LIN {X 0.253,Y -606.184,Z 1339.063,A 0.000,B 0.000,C 90.000,E1 47.391} C_DIS
LIN {X 0.399,Y -606.408,Z 1339.055,A 0.000,B 0.000,C 90.000,E1 45.810} C_DIS
LIN {X 0.066,Y -606.395,Z 1339.049,A 0.000,B 0.000,C 90.000,E1 44.798} C_DIS
LIN {X -0.075,Y -606.253,Z 1339.045,A 0.000,B 0.000,C 90.000,E1 44.028} C_DIS
LIN {X 0.206,Y -605.996,Z 1339.040,A 0.000,B 0.000,C 90.000,E1 43.218} C_DIS
LIN {X -0.072,Y -605.394,Z 1339.031,A 0.000,B 0.000,C 90.000,E1 41.676} C_DIS
LIN {X -0.161,Y -604.795,Z 1339.024,A 0.000,B 0.000,C 90.000,E1 40.378} C_DIS
LIN {X 0.075,Y -603.985,Z 1339.016,A 0.000,B 0.000,C 90.000,E1 38.785} C_DIS
LIN {X 0.122,Y -603.759,Z 1339.013,A 0.000,B 0.000,C 90.000,E1 38.257} C_DIS
LIN {X 0.089,Y -602.680,Z 1339.005,A 0.000,B 0.000,C 90.000,E1 36.950} C_DIS
LIN {X -0.224,Y -601.348,Z 1339.000,A 0.000,B 0.000,C 90.000,E1 35.931} C_DIS
LIN {X -0.077,Y -599.648,Z 1338.994,A 0.000,B 0.000,C 90.000,E1 34.865} C_DIS
LIN {X -0.395,Y -597.109,Z 1338.986,A 0.000,B 0.000,C 90.000,E1 33.579} C_DIS
LIN {X -0.042,Y -595.373,Z 1338.982,A 0.000,B 0.000,C 90.000,E1 32.752} C_DIS
LIN {X -0.025,Y -593.352,Z 1338.978,A 0.000,B 0.000,C 90.000,E1 31.957} C_DIS
LIN {X 0.082,Y -591.844,Z 1338.975,A 0.000,B 0.000,C 90.000,E1 31.416} C_DIS
LIN {X 0.258,Y -588.410,Z 1338.969,A 0.000,B 0.000,C 90.000,E1 30.335} C_DIS
LIN {X 0.204,Y -585.387,Z 1338.964,A 0.000,B 0.000,C 90.000,E1 29.539} C_DIS
LIN {X -0.037,Y -583.137,Z 1338.961,A 0.000,B 0.000,C 90.000,E1 29.027} C_DIS
LIN {X -0.212,Y -578.917,Z 1338.956,A 0.000,B 0.000,C 90.000,E1 28.103} C_DIS
LIN {X 0.212,Y -575.437,Z 1338.952,A 0.000,B 0.000,C 90.000,E1 27.385} C_DIS
LIN {X -0.253,Y -570.967,Z 1338.948,A 0.000,B 0.000,C 90.000,E1 26.616} C_DIS
LIN {X -0.161,Y -566.910,Z 1338.944,A 0.000,B 0.000,C 90.000,E1 25.924} C_DIS
LIN {X 0.139,Y -562.460,Z 1338.940,A 0.000,B 0.000,C 90.000,E1 25.207} C_DIS
LIN {X -0.057,Y -555.714,Z 1338.935,A 0.000,B 0.000,C 90.000,E1 24.259} C_DIS
LIN {X -0.045,Y -547.161,Z 1338.929,A 0.000,B 0.000,C 90.000,E1 23.153} C_DIS
LIN {X -0.036,Y -542.466,Z 1338.926,A 0.000,B 0.000,C 90.000,E1 22.589} C_DIS
LIN {X 0.115,Y -532.861,Z 1338.919,A 0.000,B 0.000,C 90.000,E1 21.482} C_DIS
LIN {X 0.055,Y -525.225,Z 1338.915,A 0.000,B 0.000,C 90.000,E1 20.663} C_DIS
LIN {X -0.228,Y -513.411,Z 1338.908,A 0.000,B 0.000,C 90.000,E1 19.450} C_DIS
LIN {X -0.010,Y -502.802,Z 1338.902,A 0.000,B 0.000,C 90.000,E1 18.308} C_DIS
LIN {X -0.186,Y -495.880,Z 1338.898,A 0.000,B 0.000,C 90.000,E1 17.638} C_DIS
LIN {X 0.077,Y -491.962,Z 1338.896,A 0.000,B 0.000,C 90.000,E1 17.221} C_DIS
LIN {X 0.076,Y -479.200,Z 1338.889,A 0.000,B 0.000,C 90.000,E1 16.024} C_DIS
LIN {X 0.163,Y -470.528,Z 1338.885,A 0.000,B 0.000,C 90.000,E1 15.190} C_DIS
LIN {X -0.090,Y -457.861,Z 1338.878,A 0.000,B 0.000,C 90.000,E1 14.008} C_DIS
LIN {X -0.116,Y -440.530,Z 1338.868,A 0.000,B 0.000,C 90.000,E1 12.299} C_DIS
LIN {X -0.086,Y -423.447,Z 1338.858,A 0.000,B 0.000,C 90.000,E1 10.489} C_DIS
LIN {X 0.042,Y -408.056,Z 1338.849,A 0.000,B 0.000,C 90.000,E1 8.746} C_DIS
LIN {X 0.112,Y -399.560,Z 1338.843,A 0.000,B 0.000,C 90.000,E1 7.757} C_DIS
LIN {X -0.011,Y -396.193,Z 1338.841,A 0.000,B 0.000,C 90.000,E1 7.352} C_DIS
LIN {X -0.095,Y -395.192,Z 1338.840,A 0.000,B 0.000,C 90.000,E1 7.182} C_DIS
LIN {X -0.159,Y -394.889,Z 1338.839,A 0.000,B 0.000,C 90.000,E1 7.125} C_DIS
LIN {X -0.197,Y -394.881,Z 1338.839,A 0.000,B 0.000,C 90.000,E1 7.125} C_DIS
LIN {X 0.156,Y -394.888,Z 1338.839,A 0.000,B 0.000,C 90.000,E1 7.068} C_DIS
LIN {X 0.119,Y -394.922,Z 1338.839,A 0.000,B 0.000,C 90.000,E1 7.068} C_DIS
LIN {X -0.088,Y -395.768,Z 1338.839,A 0.000,B 0.000,C 90.000,E1 7.004} C_DIS
LIN {X 0.079,Y -399.281,Z 1338.837,A 0.000,B 0.000,C 90.000,E1 6.663} C_DIS
LIN {X -0.111,Y -407.017,Z 1338.834,A 0.000,B 0.000,C 90.000,E1 6.144} C_DIS
LIN {X 0.037,Y -415.213,Z 1338.831,A 0.000,B 0.000,C 90.000,E1 5.568} C_DIS
LIN {X 0.038,Y -416.883,Z 1338.830,A 0.000,B 0.000,C 90.000,E1 5.454} C_DIS
LIN {X -0.059,Y -423.003,Z 1338.828,A 0.000,B 0.000,C 90.000,E1 4.992} C_DIS
LIN {X -0.215,Y -430.404,Z 1338.824,A 0.000,B 0.000,C 90.000,E1 4.359} C_DIS
LIN {X 0.191,Y -439.080,Z 1338.819,A 0.000,B 0.000,C 90.000,E1 3.440} C_DIS
LIN {X -0.097,Y -443.387,Z 1338.817,A 0.000,B 0.000,C 90.000,E1 3.037} C_DIS
LIN {X 0.196,Y -450.196,Z 1338.813,A 0.000,B 0.000,C 90.000,E1 2.236} C_DIS
LIN {X -0.176,Y -455.607,Z 1338.809,A 0.000,B 0.000,C 90.000,E1 1.661} C_DIS
LIN {X 0.189,Y -461.755,Z 1338.805,A 0.000,B 0.000,C 90.000,E1 0.859} C_DIS
LIN {X 0.147,Y -466.546,Z 1338.801,A 0.000,B 0.000,C 90.000,E1 0.229} C_DIS
LIN {X 0.070,Y -473.059,Z 1338.796,A 0.000,B 0.000,C 90.000,E1 359.312} C_DIS
LIN {X -0.233,Y -478.042,Z 1338.792,A 0.000,B 0.000,C 90.000,E1 358.568} C_DIS
LIN {X 0.005,Y -482.684,Z 1338.788,A 0.000,B 0.000,C 90.000,E1 357.764} C_DIS
LIN {X -0.217,Y -486.975,Z 1338.783,A 0.000,B 0.000,C 90.000,E1 357.020} C_DIS
LIN {X -0.048,Y -490.251,Z 1338.780,A 0.000,B 0.000,C 90.000,E1 356.388} C_DIS
LIN {X -0.173,Y -493.903,Z 1338.776,A 0.000,B 0.000,C 90.000,E1 355.641} C_DIS
LIN {X -0.093,Y -497.944,Z 1338.771,A 0.000,B 0.000,C 90.000,E1 354.723} C_DIS
LIN {X -0.099,Y -501.093,Z 1338.766,A 0.000,B 0.000,C 90.000,E1 353.970} C_DIS
LIN {X 0.187,Y -503.472,Z 1338.763,A 0.000,B 0.000,C 90.000,E1 353.337} C_DIS
LIN {X -0.014,Y -505.647,Z 1338.760,A 0.000,B 0.000,C 90.000,E1 352.761} C_DIS
LIN {X 0.195,Y -509.626,Z 1338.753,A 0.000,B 0.000,C 90.000,E1 351.546} C_DIS
LIN {X -0.008,Y -512.111,Z 1338.748,A 0.000,B 0.000,C 90.000,E1 350.679} C_DIS
LIN {X -0.125,Y -515.124,Z 1338.742,A 0.000,B 0.000,C 90.000,E1 349.511} C_DIS
LIN {X -0.180,Y -517.123,Z 1338.737,A 0.000,B 0.000,C 90.000,E1 348.634} C_DIS
LIN {X -0.221,Y -519.485,Z 1338.730,A 0.000,B 0.000,C 90.000,E1 347.465} C_DIS
LIN {X -0.114,Y -521.403,Z 1338.724,A 0.000,B 0.000,C 90.000,E1 346.284} C_DIS
LIN {X -0.110,Y -522.626,Z 1338.719,A 0.000,B 0.000,C 90.000,E1 345.408} C_DIS
LIN {X 0.031,Y -523.577,Z 1338.714,A 0.000,B 0.000,C 90.000,E1 344.519} C_DIS
LIN {X 0.181,Y -524.262,Z 1338.709,A 0.000,B 0.000,C 90.000,E1 343.630} C_DIS
LIN {X -0.012,Y -524.796,Z 1338.704,A 0.000,B 0.000,C 90.000,E1 342.779} C_DIS
LIN {X 0.146,Y -524.986,Z 1338.700,A 0.000,B 0.000,C 90.000,E1 341.891} C_DIS
LIN {X 0.131,Y -524.847,Z 1338.693,A 0.000,B 0.000,C 90.000,E1 340.732} C_DIS
LIN {X 0.119,Y -524.172,Z 1338.687,A 0.000,B 0.000,C 90.000,E1 339.571} C_DIS
LIN {X -0.067,Y -523.171,Z 1338.682,A 0.000,B 0.000,C 90.000,E1 338.720} C_DIS
LIN {X -0.231,Y -522.344,Z 1338.679,A 0.000,B 0.000,C 90.000,E1 338.156} C_DIS
LIN {X 0.086,Y -521.302,Z 1338.675,A 0.000,B 0.000,C 90.000,E1 337.539} C_DIS
LIN {X 0.240,Y -520.884,Z 1338.674,A 0.000,B 0.000,C 90.000,E1 337.230} C_DIS
LIN {X 0.211,Y -519.215,Z 1338.669,A 0.000,B 0.000,C 90.000,E1 336.357} C_DIS
LIN {X 0.164,Y -517.178,Z 1338.664,A 0.000,B 0.000,C 90.000,E1 335.485} C_DIS
LIN {X -0.039,Y -515.538,Z 1338.661,A 0.000,B 0.000,C 90.000,E1 334.921} C_DIS
LIN {X 0.088,Y -514.530,Z 1338.659,A 0.000,B 0.000,C 90.000,E1 334.613} C_DIS
LIN {X 0.260,Y -512.726,Z 1338.657,A 0.000,B 0.000,C 90.000,E1 334.152} C_DIS
LIN {X -0.087,Y -511.256,Z 1338.655,A 0.000,B 0.000,C 90.000,E1 333.896} C_DIS
LIN {X 0.021,Y -509.372,Z 1338.653,A 0.000,B 0.000,C 90.000,E1 333.589} C_DIS
LIN {X 0.072,Y -508.133,Z 1338.652,A 0.000,B 0.000,C 90.000,E1 333.435} C_DIS
LIN {X -0.106,Y -506.196,Z 1338.652,A 0.000,B 0.000,C 90.000,E1 333.307} C_DIS
LIN {X 0.011,Y -479.286,Z 1338.643,A 0.000,B 0.000,C 90.000,E1 331.691} C_DIS
LIN {X -0.186,Y -453.786,Z 1338.633,A 0.000,B 0.000,C 90.000,E1 329.999} C_DIS
LIN {X -0.103,Y -430.314,Z 1338.623,A 0.000,B 0.000,C 90.000,E1 328.201} C_DIS
LIN {X -0.021,Y -408.839,Z 1338.613,A 0.000,B 0.000,C 90.000,E1 326.342} C_DIS
LIN {X -0.250,Y -389.331,Z 1338.603,A 0.000,B 0.000,C 90.000,E1 324.482} C_DIS
LIN {X 0.072,Y -372.802,Z 1338.593,A 0.000,B 0.000,C 90.000,E1 322.637} C_DIS
LIN {X 0.038,Y -372.777,Z 1338.593,A 0.000,B 0.000,C 90.000,E1 322.637} C_DIS
LIN {X -0.181,Y -377.925,Z 1338.565,A 0.000,B 0.000,C 90.000,E1 317.634} C_DIS
LIN {X 0.101,Y -378.518,Z 1338.561,A 0.000,B 0.000,C 90.000,E1 316.863} C_DIS
LIN {X 0.124,Y -384.530,Z 1338.528,A 0.000,B 0.000,C 90.000,E1 311.067} C_DIS
LIN {X 0.169,Y -384.938,Z 1338.526,A 0.000,B 0.000,C 90.000,E1 310.701} C_DIS
LIN {X -0.203,Y -390.704,Z 1338.495,A 0.000,B 0.000,C 90.000,E1 305.025} C_DIS
LIN {X 0.186,Y -391.200,Z 1338.492,A 0.000,B 0.000,C 90.000,E1 304.612} C_DIS
LIN {X -0.008,Y -396.914,Z 1338.459,A 0.000,B 0.000,C 90.000,E1 298.615} C_DIS
LIN {X 0.092,Y -398.138,Z 1338.447,A 0.000,B 0.000,C 90.000,E1 296.488} C_DIS
LIN {X 0.003,Y -401.640,Z 1338.426,A 0.000,B 0.000,C 90.000,E1 292.642} C_DIS
LIN {X 0.140,Y -404.716,Z 1338.395,A 0.000,B 0.000,C 90.000,E1 287.040} C_DIS
LIN {X 0.142,Y -406.138,Z 1338.364,A 0.000,B 0.000,C 90.000,E1 281.478} C_DIS
LIN {X -0.163,Y -405.688,Z 1338.333,A 0.000,B 0.000,C 90.000,E1 275.967} C_DIS
LIN {X -0.093,Y -403.573,Z 1338.306,A 0.000,B 0.000,C 90.000,E1 271.088} C_DIS
LIN {X -0.158,Y -403.236,Z 1338.302,A 0.000,B 0.000,C 90.000,E1 270.401} C_DIS
LIN {X 0.080,Y -399.090,Z 1338.273,A 0.000,B 0.000,C 90.000,E1 265.122} C_DIS
LIN {X 0.022,Y -398.849,Z 1338.271,A 0.000,B 0.000,C 90.000,E1 264.780} C_DIS
LIN {X -0.080,Y -393.334,Z 1338.244,A 0.000,B 0.000,C 90.000,E1 259.859} C_DIS
LIN {X -0.157,Y -392.752,Z 1338.240,A 0.000,B 0.000,C 90.000,E1 259.162} C_DIS
LIN {X -0.079,Y -386.305,Z 1338.214,A 0.000,B 0.000,C 90.000,E1 254.519} C_DIS
LIN {X -0.007,Y -385.202,Z 1338.208,A 0.000,B 0.000,C 90.000,E1 253.433} C_DIS
LIN {X -0.076,Y -383.985,Z 1338.204,A 0.000,B 0.000,C 90.000,E1 252.725} C_DIS
LIN {X 0.104,Y -377.428,Z 1338.180,A 0.000,B 0.000,C 90.000,E1 248.358} C_DIS
LIN {X -0.009,Y -376.156,Z 1338.174,A 0.000,B 0.000,C 90.000,E1 247.283} C_DIS
LIN {X 0.162,Y -368.322,Z 1338.147,A 0.000,B 0.000,C 90.000,E1 242.487} C_DIS
LIN {X -0.121,Y -366.461,Z 1338.139,A 0.000,B 0.000,C 90.000,E1 241.051} C_DIS
LIN {X -0.037,Y -365.910,Z 1338.137,A 0.000,B 0.000,C 90.000,E1 240.667} C_DIS
LIN {X 0.053,Y -359.095,Z 1338.114,A 0.000,B 0.000,C 90.000,E1 236.548} C_DIS
LIN {X 0.139,Y -356.241,Z 1338.102,A 0.000,B 0.000,C 90.000,E1 234.276} C_DIS
LIN {X 0.070,Y -355.710,Z 1338.100,A 0.000,B 0.000,C 90.000,E1 233.909} C_DIS
LIN {X -0.126,Y -348.702,Z 1338.074,A 0.000,B 0.000,C 90.000,E1 229.380} C_DIS
LIN {X -0.052,Y -346.112,Z 1338.062,A 0.000,B 0.000,C 90.000,E1 227.067} C_DIS
LIN {X 0.045,Y -342.133,Z 1338.047,A 0.000,B 0.000,C 90.000,E1 224.352} C_DIS
LIN {X -0.030,Y -339.366,Z 1338.034,A 0.000,B 0.000,C 90.000,E1 222.081} C_DIS
LIN {X -0.047,Y -339.370,Z 1338.034,A 0.000,B 0.000,C 90.000,E1 222.081} C_DIS
LIN {X -0.114,Y -354.911,Z 1338.022,A 0.000,B 0.000,C 90.000,E1 219.930} C_DIS
LIN {X 0.201,Y -372.383,Z 1338.010,A 0.000,B 0.000,C 90.000,E1 217.729} C_DIS
LIN {X -0.033,Y -390.341,Z 1337.999,A 0.000,B 0.000,C 90.000,E1 215.804} C_DIS
LIN {X 0.009,Y -410.273,Z 1337.988,A 0.000,B 0.000,C 90.000,E1 213.865} C_DIS
LIN {X -0.172,Y -432.208,Z 1337.978,A 0.000,B 0.000,C 90.000,E1 212.005} C_DIS
LIN {X -0.113,Y -444.925,Z 1337.972,A 0.000,B 0.000,C 90.000,E1 211.003} C_DIS
LIN {X -0.011,Y -446.772,Z 1337.971,A 0.000,B 0.000,C 90.000,E1 210.747} C_DIS
LIN {X 0.053,Y -448.264,Z 1337.969,A 0.000,B 0.000,C 90.000,E1 210.413} C_DIS
LIN {X 0.127,Y -449.354,Z 1337.967,A 0.000,B 0.000,C 90.000,E1 210.079} C_DIS
LIN {X -0.188,Y -450.226,Z 1337.965,A 0.000,B 0.000,C 90.000,E1 209.795} C_DIS
LIN {X -0.028,Y -451.560,Z 1337.962,A 0.000,B 0.000,C 90.000,E1 209.127} C_DIS
LIN {X 0.011,Y -453.019,Z 1337.956,A 0.000,B 0.000,C 90.000,E1 208.153} C_DIS
LIN {X -0.178,Y -456.849,Z 1337.940,A 0.000,B 0.000,C 90.000,E1 205.283} C_DIS
LIN {X 0.148,Y -458.996,Z 1337.932,A 0.000,B 0.000,C 90.000,E1 203.643} C_DIS
LIN {X -0.096,Y -461.026,Z 1337.923,A 0.000,B 0.000,C 90.000,E1 202.078} C_DIS
LIN {X 0.023,Y -462.739,Z 1337.916,A 0.000,B 0.000,C 90.000,E1 200.791} C_DIS
LIN {X -0.195,Y -465.367,Z 1337.903,A 0.000,B 0.000,C 90.000,E1 198.598} C_DIS
LIN {X -0.166,Y -466.928,Z 1337.896,A 0.000,B 0.000,C 90.000,E1 197.330} C_DIS
LIN {X 0.131,Y -468.579,Z 1337.887,A 0.000,B 0.000,C 90.000,E1 195.717} C_DIS
LIN {X -0.117,Y -470.221,Z 1337.879,A 0.000,B 0.000,C 90.000,E1 194.175} C_DIS
LIN {X 0.187,Y -471.582,Z 1337.872,A 0.000,B 0.000,C 90.000,E1 192.883} C_DIS
LIN {X 0.004,Y -473.943,Z 1337.860,A 0.000,B 0.000,C 90.000,E1 190.715} C_DIS
LIN {X -0.132,Y -475.948,Z 1337.849,A 0.000,B 0.000,C 90.000,E1 188.859} C_DIS
LIN {X 0.098,Y -477.102,Z 1337.842,A 0.000,B 0.000,C 90.000,E1 187.587} C_DIS
LIN {X -0.129,Y -478.224,Z 1337.835,A 0.000,B 0.000,C 90.000,E1 186.372} C_DIS
LIN {X 0.079,Y -479.080,Z 1337.828,A 0.000,B 0.000,C 90.000,E1 185.106} C_DIS
LIN {X -0.178,Y -479.750,Z 1337.822,A 0.000,B 0.000,C 90.000,E1 183.898} C_DIS
LIN {X 0.020,Y -480.187,Z 1337.815,A 0.000,B 0.000,C 90.000,E1 182.636} C_DIS
LIN {X 0.224,Y -480.285,Z 1337.808,A 0.000,B 0.000,C 90.000,E1 181.375} C_DIS
LIN {X 0.129,Y -480.272,Z 1337.803,A 0.000,B 0.000,C 90.000,E1 180.458} C_DIS
LIN {X 0.131,Y -479.730,Z 1337.794,A 0.000,B 0.000,C 90.000,E1 178.912} C_DIS
LIN {X -0.151,Y -479.049,Z 1337.787,A 0.000,B 0.000,C 90.000,E1 177.707} C_DIS
LIN {X 0.236,Y -478.332,Z 1337.782,A 0.000,B 0.000,C 90.000,E1 176.731} C_DIS
LIN {X 0.140,Y -477.340,Z 1337.777,A 0.000,B 0.000,C 90.000,E1 175.812} C_DIS
LIN {X 0.029,Y -476.118,Z 1337.772,A 0.000,B 0.000,C 90.000,E1 174.894} C_DIS
LIN {X 0.118,Y -475.094,Z 1337.768,A 0.000,B 0.000,C 90.000,E1 174.261} C_DIS
LIN {X 0.198,Y -473.942,Z 1337.765,A 0.000,B 0.000,C 90.000,E1 173.628} C_DIS
LIN {X 0.093,Y -471.839,Z 1337.760,A 0.000,B 0.000,C 90.000,E1 172.704} C_DIS
LIN {X 0.208,Y -469.926,Z 1337.756,A 0.000,B 0.000,C 90.000,E1 172.064} C_DIS
LIN {X 0.058,Y -466.558,Z 1337.751,A 0.000,B 0.000,C 90.000,E1 171.141} C_DIS
LIN {X -0.035,Y -464.383,Z 1337.748,A 0.000,B 0.000,C 90.000,E1 170.679} C_DIS
LIN {X 0.024,Y -461.187,Z 1337.745,A 0.000,B 0.000,C 90.000,E1 170.038} C_DIS
LIN {X -0.162,Y -455.604,Z 1337.739,A 0.000,B 0.000,C 90.000,E1 169.106} C_DIS
LIN {X -0.020,Y -450.527,Z 1337.735,A 0.000,B 0.000,C 90.000,E1 168.285} C_DIS
LIN {X -0.025,Y -440.963,Z 1337.727,A 0.000,B 0.000,C 90.000,E1 166.825} C_DIS
LIN {X -0.106,Y -432.409,Z 1337.719,A 0.000,B 0.000,C 90.000,E1 165.519} C_DIS
LIN {X 0.098,Y -423.894,Z 1337.712,A 0.000,B 0.000,C 90.000,E1 164.157} C_DIS
LIN {X -0.145,Y -420.962,Z 1337.709,A 0.000,B 0.000,C 90.000,E1 163.685} C_DIS
LIN {X 0.070,Y -418.452,Z 1337.706,A 0.000,B 0.000,C 90.000,E1 163.015} C_DIS
LIN {X 0.031,Y -417.875,Z 1337.705,A 0.000,B 0.000,C 90.000,E1 162.851} C_DIS
LIN {X 0.114,Y -417.753,Z 1337.704,A 0.000,B 0.000,C 90.000,E1 162.670} C_DIS
LIN {X 0.148,Y -417.693,Z 1337.701,A 0.000,B 0.000,C 90.000,E1 162.181} C_DIS
LIN {X 0.109,Y -417.716,Z 1337.701,A 0.000,B 0.000,C 90.000,E1 162.181} C_DIS
LIN {X -0.198,Y -418.731,Z 1337.700,A 0.000,B 0.000,C 90.000,E1 162.000} C_DIS
LIN {X 0.086,Y -421.669,Z 1337.698,A 0.000,B 0.000,C 90.000,E1 161.638} C_DIS
LIN {X 0.067,Y -423.536,Z 1337.697,A 0.000,B 0.000,C 90.000,E1 161.402} C_DIS
LIN {X 0.254,Y -432.248,Z 1337.693,A 0.000,B 0.000,C 90.000,E1 160.604} C_DIS
LIN {X -0.113,Y -448.000,Z 1337.686,A 0.000,B 0.000,C 90.000,E1 159.444} C_DIS
LIN {X 0.128,Y -460.353,Z 1337.681,A 0.000,B 0.000,C 90.000,E1 158.465} C_DIS
LIN {X 0.269,Y -468.108,Z 1337.677,A 0.000,B 0.000,C 90.000,E1 157.847} C_DIS
LIN {X 0.269,Y -477.193,Z 1337.673,A 0.000,B 0.000,C 90.000,E1 157.102} C_DIS
LIN {X 0.126,Y -481.670,Z 1337.671,A 0.000,B 0.000,C 90.000,E1 156.741} C_DIS
LIN {X 0.053,Y -487.508,Z 1337.668,A 0.000,B 0.000,C 90.000,E1 156.230} C_DIS
LIN {X -0.275,Y -494.447,Z 1337.664,A 0.000,B 0.000,C 90.000,E1 155.613} C_DIS
LIN {X -0.152,Y -499.988,Z 1337.661,A 0.000,B 0.000,C 90.000,E1 155.049} C_DIS
LIN {X 0.132,Y -506.591,Z 1337.658,A 0.000,B 0.000,C 90.000,E1 154.332} C_DIS
LIN {X -0.015,Y -512.927,Z 1337.654,A 0.000,B 0.000,C 90.000,E1 153.640} C_DIS
LIN {X 0.094,Y -517.761,Z 1337.650,A 0.000,B 0.000,C 90.000,E1 153.050} C_DIS
LIN {X -0.115,Y -522.268,Z 1337.647,A 0.000,B 0.000,C 90.000,E1 152.487} C_DIS
LIN {X 0.106,Y -525.392,Z 1337.645,A 0.000,B 0.000,C 90.000,E1 152.025} C_DIS
LIN {X 0.197,Y -529.034,Z 1337.641,A 0.000,B 0.000,C 90.000,E1 151.435} C_DIS
LIN {X 0.057,Y -532.019,Z 1337.638,A 0.000,B 0.000,C 90.000,E1 150.873} C_DIS
LIN {X 0.021,Y -533.358,Z 1337.637,A 0.000,B 0.000,C 90.000,E1 150.589} C_DIS
LIN {X 0.168,Y -535.696,Z 1337.633,A 0.000,B 0.000,C 90.000,E1 149.999} C_DIS
LIN {X -0.134,Y -537.738,Z 1337.630,A 0.000,B 0.000,C 90.000,E1 149.459} C_DIS
LIN {X 0.045,Y -540.275,Z 1337.625,A 0.000,B 0.000,C 90.000,E1 148.584} C_DIS
LIN {X 0.239,Y -541.833,Z 1337.622,A 0.000,B 0.000,C 90.000,E1 147.995} C_DIS
LIN {X 0.004,Y -543.833,Z 1337.618,A 0.000,B 0.000,C 90.000,E1 147.168} C_DIS
LIN {X 0.280,Y -546.008,Z 1337.611,A 0.000,B 0.000,C 90.000,E1 146.008} C_DIS
LIN {X 0.088,Y -547.311,Z 1337.607,A 0.000,B 0.000,C 90.000,E1 145.182} C_DIS
LIN {X -0.047,Y -548.611,Z 1337.600,A 0.000,B 0.000,C 90.000,E1 144.069} C_DIS
LIN {X 0.156,Y -549.612,Z 1337.594,A 0.000,B 0.000,C 90.000,E1 142.924} C_DIS
LIN {X 0.107,Y -550.845,Z 1337.583,A 0.000,B 0.000,C 90.000,E1 140.964} C_DIS
LIN {X -0.152,Y -551.367,Z 1337.579,A 0.000,B 0.000,C 90.000,E1 140.150} C_DIS
LIN {X -0.178,Y -553.325,Z 1337.565,A 0.000,B 0.000,C 90.000,E1 137.634} C_DIS
LIN {X -0.103,Y -554.134,Z 1337.562,A 0.000,B 0.000,C 90.000,E1 137.067} C_DIS
LIN {X 0.114,Y -554.328,Z 1337.561,A 0.000,B 0.000,C 90.000,E1 136.905} C_DIS
LIN {X 0.169,Y -555.407,Z 1337.559,A 0.000,B 0.000,C 90.000,E1 136.620} C_DIS
LIN {X 0.068,Y -555.741,Z 1337.558,A 0.000,B 0.000,C 90.000,E1 136.500} C_DIS
LIN {X 0.026,Y -555.787,Z 1337.558,A 0.000,B 0.000,C 90.000,E1 136.500} C_DIS
LIN {X -0.160,Y -556.939,Z 1337.558,A 0.000,B 0.000,C 90.000,E1 136.458} C_DIS
LIN {X 0.029,Y -564.205,Z 1337.557,A 0.000,B 0.000,C 90.000,E1 136.215} C_DIS
LIN {X 0.238,Y -569.544,Z 1337.556,A 0.000,B 0.000,C 90.000,E1 136.053} C_DIS
LIN {X -0.241,Y -575.649,Z 1337.555,A 0.000,B 0.000,C 90.000,E1 135.891} C_DIS
LIN {X 0.120,Y -578.484,Z 1337.554,A 0.000,B 0.000,C 90.000,E1 135.729} C_DIS
LIN {X 0.030,Y -584.123,Z 1337.552,A 0.000,B 0.000,C 90.000,E1 135.405} C_DIS
LIN {X -0.283,Y -587.197,Z 1337.551,A 0.000,B 0.000,C 90.000,E1 135.243} C_DIS
LIN {X -0.052,Y -591.466,Z 1337.550,A 0.000,B 0.000,C 90.000,E1 134.919} C_DIS
LIN {X -0.007,Y -598.522,Z 1337.546,A 0.000,B 0.000,C 90.000,E1 134.352} C_DIS
LIN {X 0.142,Y -602.051,Z 1337.545,A 0.000,B 0.000,C 90.000,E1 134.028} C_DIS
LIN {X 0.138,Y -607.076,Z 1337.542,A 0.000,B 0.000,C 90.000,E1 133.542} C_DIS
LIN {X -0.074,Y -611.948,Z 1337.539,A 0.000,B 0.000,C 90.000,E1 133.056} C_DIS
LIN {X -0.303,Y -615.513,Z 1337.537,A 0.000,B 0.000,C 90.000,E1 132.690} C_DIS
LIN {X 0.183,Y -620.944,Z 1337.533,A 0.000,B 0.000,C 90.000,E1 132.000} C_DIS
LIN {X 0.211,Y -627.072,Z 1337.529,A 0.000,B 0.000,C 90.000,E1 131.229} C_DIS
LIN {X -0.055,Y -631.010,Z 1337.526,A 0.000,B 0.000,C 90.000,E1 130.744} C_DIS
LIN {X -0.345,Y -636.582,Z 1337.522,A 0.000,B 0.000,C 90.000,E1 130.011} C_DIS
LIN {X -0.177,Y -642.849,Z 1337.517,A 0.000,B 0.000,C 90.000,E1 129.116} C_DIS
LIN {X 0.158,Y -647.902,Z 1337.513,A 0.000,B 0.000,C 90.000,E1 128.338} C_DIS
LIN {X 0.042,Y -652.812,Z 1337.509,A 0.000,B 0.000,C 90.000,E1 127.604} C_DIS
LIN {X -0.094,Y -658.940,Z 1337.504,A 0.000,B 0.000,C 90.000,E1 126.629} C_DIS
LIN {X 0.026,Y -663.200,Z 1337.499,A 0.000,B 0.000,C 90.000,E1 125.884} C_DIS
LIN {X 0.085,Y -665.835,Z 1337.497,A 0.000,B 0.000,C 90.000,E1 125.391} C_DIS
LIN {X -0.265,Y -669.292,Z 1337.493,A 0.000,B 0.000,C 90.000,E1 124.692} C_DIS
LIN {X -0.171,Y -671.465,Z 1337.490,A 0.000,B 0.000,C 90.000,E1 124.199} C_DIS
LIN {X 0.088,Y -674.303,Z 1337.486,A 0.000,B 0.000,C 90.000,E1 123.452} C_DIS
LIN {X -0.190,Y -676.696,Z 1337.482,A 0.000,B 0.000,C 90.000,E1 122.752} C_DIS
LIN {X 0.122,Y -678.819,Z 1337.478,A 0.000,B 0.000,C 90.000,E1 122.005} C_DIS
LIN {X 0.101,Y -680.707,Z 1337.474,A 0.000,B 0.000,C 90.000,E1 121.288} C_DIS
LIN {X -0.132,Y -682.319,Z 1337.470,A 0.000,B 0.000,C 90.000,E1 120.590} C_DIS
LIN {X -0.115,Y -683.639,Z 1337.466,A 0.000,B 0.000,C 90.000,E1 119.873} C_DIS
LIN {X -0.079,Y -684.623,Z 1337.462,A 0.000,B 0.000,C 90.000,E1 119.155} C_DIS
LIN {X -0.250,Y -685.066,Z 1337.459,A 0.000,B 0.000,C 90.000,E1 118.693} C_DIS
LIN {X -0.200,Y -685.514,Z 1337.455,A 0.000,B 0.000,C 90.000,E1 117.975} C_DIS
LIN {X 0.073,Y -685.669,Z 1337.450,A 0.000,B 0.000,C 90.000,E1 117.001} C_DIS
LIN {X 0.119,Y -685.571,Z 1337.446,A 0.000,B 0.000,C 90.000,E1 116.283} C_DIS
LIN {X -0.139,Y -685.180,Z 1337.442,A 0.000,B 0.000,C 90.000,E1 115.591} C_DIS
LIN {X 0.296,Y -684.734,Z 1337.440,A 0.000,B 0.000,C 90.000,E1 115.079} C_DIS
LIN {X -0.181,Y -684.006,Z 1337.437,A 0.000,B 0.000,C 90.000,E1 114.643} C_DIS
LIN {X -0.035,Y -682.924,Z 1337.434,A 0.000,B 0.000,C 90.000,E1 114.155} C_DIS
LIN {X -0.141,Y -680.402,Z 1337.431,A 0.000,B 0.000,C 90.000,E1 113.567} C_DIS
LIN {X -0.040,Y -679.588,Z 1337.430,A 0.000,B 0.000,C 90.000,E1 113.439} C_DIS
LIN {X -0.017,Y -676.352,Z 1337.428,A 0.000,B 0.000,C 90.000,E1 113.078} C_DIS
LIN {X 0.077,Y -675.321,Z 1337.428,A 0.000,B 0.000,C 90.000,E1 112.950} C_DIS
LIN {X 0.167,Y -673.832,Z 1337.427,A 0.000,B 0.000,C 90.000,E1 112.823} C_DIS
LIN {X -0.131,Y -669.957,Z 1337.426,A 0.000,B 0.000,C 90.000,E1 112.642} C_DIS
LIN {X 0.135,Y -665.122,Z 1337.424,A 0.000,B 0.000,C 90.000,E1 112.386} C_DIS
LIN {X -0.182,Y -660.200,Z 1337.424,A 0.000,B 0.000,C 90.000,E1 112.259} C_DIS
LIN {X -0.182,Y -657.989,Z 1337.423,A 0.000,B 0.000,C 90.000,E1 112.206} C_DIS
LIN {X -0.189,Y -643.923,Z 1337.422,A 0.000,B 0.000,C 90.000,E1 111.972} C_DIS
LIN {X -0.160,Y -640.586,Z 1337.422,A 0.000,B 0.000,C 90.000,E1 111.897} C_DIS
LIN {X -0.214,Y -640.430,Z 1337.422,A 0.000,B 0.000,C 90.000,E1 111.897} C_DIS
LIN {X -0.158,Y -642.482,Z 1337.420,A 0.000,B 0.000,C 90.000,E1 111.589} C_DIS
LIN {X -0.001,Y -647.833,Z 1337.416,A 0.000,B 0.000,C 90.000,E1 110.918} C_DIS
LIN {X -0.081,Y -651.611,Z 1337.413,A 0.000,B 0.000,C 90.000,E1 110.429} C_DIS
LIN {X -0.094,Y -655.667,Z 1337.410,A 0.000,B 0.000,C 90.000,E1 109.812} C_DIS
LIN {X -0.128,Y -658.482,Z 1337.407,A 0.000,B 0.000,C 90.000,E1 109.322} C_DIS
LIN {X -0.309,Y -661.461,Z 1337.404,A 0.000,B 0.000,C 90.000,E1 108.725} C_DIS
LIN {X 0.221,Y -664.651,Z 1337.400,A 0.000,B 0.000,C 90.000,E1 107.946} C_DIS
LIN {X 0.154,Y -667.487,Z 1337.396,A 0.000,B 0.000,C 90.000,E1 107.221} C_DIS
LIN {X 0.110,Y -670.028,Z 1337.392,A 0.000,B 0.000,C 90.000,E1 106.496} C_DIS
LIN {X -0.033,Y -671.559,Z 1337.389,A 0.000,B 0.000,C 90.000,E1 106.024} C_DIS
LIN {X -0.046,Y -673.460,Z 1337.385,A 0.000,B 0.000,C 90.000,E1 105.300} C_DIS
LIN {X -0.223,Y -675.078,Z 1337.381,A 0.000,B 0.000,C 90.000,E1 104.592} C_DIS
LIN {X -0.278,Y -675.580,Z 1337.380,A 0.000,B 0.000,C 90.000,E1 104.356} C_DIS
LIN {X 0.225,Y -676.640,Z 1337.376,A 0.000,B 0.000,C 90.000,E1 103.592} C_DIS
LIN {X 0.128,Y -677.179,Z 1337.373,A 0.000,B 0.000,C 90.000,E1 103.119} C_DIS
LIN {X -0.013,Y -677.434,Z 1337.369,A 0.000,B 0.000,C 90.000,E1 102.411} C_DIS
LIN {X -0.248,Y -677.496,Z 1337.366,A 0.000,B 0.000,C 90.000,E1 101.951} C_DIS
LIN {X -0.341,Y -677.368,Z 1337.364,A 0.000,B 0.000,C 90.000,E1 101.478} C_DIS
LIN {X 0.227,Y -676.957,Z 1337.361,A 0.000,B 0.000,C 90.000,E1 100.950} C_DIS
LIN {X -0.053,Y -675.982,Z 1337.357,A 0.000,B 0.000,C 90.000,E1 100.254} C_DIS
LIN {X -0.166,Y -675.031,Z 1337.354,A 0.000,B 0.000,C 90.000,E1 99.782} C_DIS
LIN {X 0.266,Y -673.879,Z 1337.352,A 0.000,B 0.000,C 90.000,E1 99.265} C_DIS
LIN {X 0.030,Y -672.325,Z 1337.349,A 0.000,B 0.000,C 90.000,E1 98.803} C_DIS
LIN {X -0.290,Y -669.500,Z 1337.345,A 0.000,B 0.000,C 90.000,E1 98.106} C_DIS
LIN {X 0.023,Y -666.218,Z 1337.341,A 0.000,B 0.000,C 90.000,E1 97.352} C_DIS
LIN {X -0.256,Y -663.843,Z 1337.338,A 0.000,B 0.000,C 90.000,E1 96.891} C_DIS
LIN {X -0.085,Y -660.006,Z 1337.334,A 0.000,B 0.000,C 90.000,E1 96.144} C_DIS
LIN {X 0.112,Y -655.569,Z 1337.330,A 0.000,B 0.000,C 90.000,E1 95.391} C_DIS
LIN {X -0.233,Y -652.484,Z 1337.327,A 0.000,B 0.000,C 90.000,E1 94.935} C_DIS
LIN {X -0.061,Y -648.166,Z 1337.324,A 0.000,B 0.000,C 90.000,E1 94.302} C_DIS
LIN {X 0.185,Y -644.501,Z 1337.321,A 0.000,B 0.000,C 90.000,E1 93.784} C_DIS
LIN {X -0.276,Y -640.519,Z 1337.318,A 0.000,B 0.000,C 90.000,E1 93.326} C_DIS
LIN {X -0.086,Y -636.047,Z 1337.316,A 0.000,B 0.000,C 90.000,E1 92.808} C_DIS
LIN {X 0.034,Y -629.843,Z 1337.312,A 0.000,B 0.000,C 90.000,E1 92.178} C_DIS
LIN {X -0.064,Y -618.494,Z 1337.306,A 0.000,B 0.000,C 90.000,E1 91.088} C_DIS
LIN {X -0.228,Y -612.984,Z 1337.303,A 0.000,B 0.000,C 90.000,E1 90.630} C_DIS
LIN {X -0.229,Y -610.251,Z 1337.302,A 0.000,B 0.000,C 90.000,E1 90.401} C_DIS
LIN {X -0.234,Y -608.680,Z 1337.302,A 0.000,B 0.000,C 90.000,E1 90.286} C_DIS
LIN {X -0.267,Y -602.169,Z 1337.299,A 0.000,B 0.000,C 90.000,E1 89.885} C_DIS
LIN {X 0.250,Y -595.008,Z 1337.297,A 0.000,B 0.000,C 90.000,E1 89.484} C_DIS
LIN {X 0.077,Y -587.859,Z 1337.296,A 0.000,B 0.000,C 90.000,E1 89.198} C_DIS
LIN {X -0.275,Y -582.624,Z 1337.294,A 0.000,B 0.000,C 90.000,E1 89.026} C_DIS
LIN {X 0.017,Y -578.234,Z 1337.293,A 0.000,B 0.000,C 90.000,E1 88.797} C_DIS
LIN {X -0.176,Y -576.884,Z 1337.293,A 0.000,B 0.000,C 90.000,E1 88.740} C_DIS
LIN {X -0.068,Y -573.417,Z 1337.291,A 0.000,B 0.000,C 90.000,E1 88.453} C_DIS
LIN {X -0.279,Y -573.242,Z 1337.291,A 0.000,B 0.000,C 90.000,E1 88.453} C_DIS
LIN {X 0.258,Y -573.218,Z 1337.291,A 0.000,B 0.000,C 90.000,E1 88.396} C_DIS
LIN {X -0.236,Y -572.514,Z 1337.290,A 0.000,B 0.000,C 90.000,E1 88.165} C_DIS
LIN {X -0.022,Y -572.470,Z 1337.287,A 0.000,B 0.000,C 90.000,E1 87.593} C_DIS
LIN {X -0.256,Y -575.018,Z 1337.271,A 0.000,B 0.000,C 90.000,E1 84.894} C_DIS
LIN {X -0.070,Y -577.511,Z 1337.260,A 0.000,B 0.000,C 90.000,E1 82.704} C_DIS
LIN {X -0.318,Y -579.149,Z 1337.252,A 0.000,B 0.000,C 90.000,E1 81.376} C_DIS
LIN {X -0.224,Y -581.103,Z 1337.243,A 0.000,B 0.000,C 90.000,E1 79.746} C_DIS
LIN {X -0.208,Y -582.504,Z 1337.235,A 0.000,B 0.000,C 90.000,E1 78.398} C_DIS
LIN {X 0.041,Y -583.562,Z 1337.229,A 0.000,B 0.000,C 90.000,E1 77.297} C_DIS
LIN {X -0.099,Y -584.904,Z 1337.221,A 0.000,B 0.000,C 90.000,E1 75.700} C_DIS
LIN {X -0.209,Y -585.989,Z 1337.212,A 0.000,B 0.000,C 90.000,E1 74.102} C_DIS
LIN {X -0.052,Y -586.767,Z 1337.206,A 0.000,B 0.000,C 90.000,E1 73.015} C_DIS
LIN {X 0.124,Y -588.132,Z 1337.194,A 0.000,B 0.000,C 90.000,E1 70.859} C_DIS
LIN {X -0.274,Y -589.239,Z 1337.183,A 0.000,B 0.000,C 90.000,E1 69.028} C_DIS
LIN {X 0.017,Y -590.097,Z 1337.176,A 0.000,B 0.000,C 90.000,E1 67.667} C_DIS
LIN {X 0.216,Y -591.211,Z 1337.167,A 0.000,B 0.000,C 90.000,E1 66.049} C_DIS
LIN {X 0.243,Y -592.173,Z 1337.160,A 0.000,B 0.000,C 90.000,E1 64.717} C_DIS
LIN {X 0.193,Y -593.321,Z 1337.151,A 0.000,B 0.000,C 90.000,E1 63.127} C_DIS
LIN {X -0.370,Y -595.261,Z 1337.138,A 0.000,B 0.000,C 90.000,E1 60.795} C_DIS
LIN {X -0.202,Y -597.331,Z 1337.126,A 0.000,B 0.000,C 90.000,E1 58.663} C_DIS
LIN {X 0.198,Y -598.948,Z 1337.117,A 0.000,B 0.000,C 90.000,E1 57.041} C_DIS
LIN {X -0.127,Y -600.843,Z 1337.107,A 0.000,B 0.000,C 90.000,E1 55.229} C_DIS
LIN {X -0.072,Y -602.149,Z 1337.099,A 0.000,B 0.000,C 90.000,E1 53.909} C_DIS
LIN {X 0.353,Y -603.351,Z 1337.092,A 0.000,B 0.000,C 90.000,E1 52.557} C_DIS
LIN {X 0.057,Y -604.106,Z 1337.086,A 0.000,B 0.000,C 90.000,E1 51.537} C_DIS
LIN {X 0.027,Y -605.017,Z 1337.079,A 0.000,B 0.000,C 90.000,E1 50.231} C_DIS
LIN {X -0.125,Y -605.477,Z 1337.075,A 0.000,B 0.000,C 90.000,E1 49.461} C_DIS
LIN {X -0.206,Y -605.945,Z 1337.068,A 0.000,B 0.000,C 90.000,E1 48.162} C_DIS
LIN {X -0.342,Y -606.102,Z 1337.063,A 0.000,B 0.000,C 90.000,E1 47.391} C_DIS
LIN {X -0.197,Y -606.324,Z 1337.054,A 0.000,B 0.000,C 90.000,E1 45.810} C_DIS
LIN {X -0.102,Y -606.303,Z 1337.049,A 0.000,B 0.000,C 90.000,E1 44.757} C_DIS
LIN {X -0.008,Y -606.084,Z 1337.043,A 0.000,B 0.000,C 90.000,E1 43.704} C_DIS
LIN {X 0.126,Y -605.492,Z 1337.034,A 0.000,B 0.000,C 90.000,E1 42.123} C_DIS
LIN {X 0.238,Y -605.094,Z 1337.028,A 0.000,B 0.000,C 90.000,E1 41.067} C_DIS
LIN {X 0.011,Y -604.321,Z 1337.020,A 0.000,B 0.000,C 90.000,E1 39.519} C_DIS
LIN {X -0.106,Y -603.663,Z 1337.012,A 0.000,B 0.000,C 90.000,E1 38.222} C_DIS
LIN {X 0.329,Y -602.617,Z 1337.005,A 0.000,B 0.000,C 90.000,E1 36.870} C_DIS
LIN {X -0.090,Y -600.860,Z 1336.998,A 0.000,B 0.000,C 90.000,E1 35.598} C_DIS
LIN {X 0.054,Y -599.026,Z 1336.992,A 0.000,B 0.000,C 90.000,E1 34.532} C_DIS
LIN {X -0.171,Y -596.979,Z 1336.986,A 0.000,B 0.000,C 90.000,E1 33.499} C_DIS
LIN {X -0.044,Y -595.878,Z 1336.983,A 0.000,B 0.000,C 90.000,E1 32.959} C_DIS
LIN {X 0.191,Y -593.204,Z 1336.977,A 0.000,B 0.000,C 90.000,E1 31.878} C_DIS
LIN {X 0.294,Y -591.665,Z 1336.974,A 0.000,B 0.000,C 90.000,E1 31.337} C_DIS
LIN {X -0.231,Y -589.151,Z 1336.970,A 0.000,B 0.000,C 90.000,E1 30.590} C_DIS
LIN {X 0.232,Y -586.207,Z 1336.965,A 0.000,B 0.000,C 90.000,E1 29.745} C_DIS
LIN {X 0.281,Y -584.104,Z 1336.962,A 0.000,B 0.000,C 90.000,E1 29.205} C_DIS
LIN {X -0.097,Y -580.520,Z 1336.958,A 0.000,B 0.000,C 90.000,E1 28.437} C_DIS
LIN {X -0.094,Y -577.949,Z 1336.955,A 0.000,B 0.000,C 90.000,E1 27.897} C_DIS
LIN {X 0.127,Y -575.145,Z 1336.952,A 0.000,B 0.000,C 90.000,E1 27.334} C_DIS
LIN {X -0.164,Y -569.864,Z 1336.947,A 0.000,B 0.000,C 90.000,E1 26.411} C_DIS
LIN {X -0.084,Y -565.656,Z 1336.943,A 0.000,B 0.000,C 90.000,E1 25.720} C_DIS
LIN {X 0.056,Y -562.052,Z 1336.940,A 0.000,B 0.000,C 90.000,E1 25.155} C_DIS
LIN {X -0.139,Y -555.288,Z 1336.934,A 0.000,B 0.000,C 90.000,E1 24.207} C_DIS
LIN {X -0.035,Y -546.532,Z 1336.928,A 0.000,B 0.000,C 90.000,E1 23.078} C_DIS
LIN {X 0.097,Y -543.043,Z 1336.926,A 0.000,B 0.000,C 90.000,E1 22.642} C_DIS
LIN {X -0.177,Y -533.041,Z 1336.920,A 0.000,B 0.000,C 90.000,E1 21.535} C_DIS
LIN {X 0.059,Y -525.213,Z 1336.915,A 0.000,B 0.000,C 90.000,E1 20.663} C_DIS
LIN {X 0.089,Y -511.947,Z 1336.907,A 0.000,B 0.000,C 90.000,E1 19.268} C_DIS
LIN {X 0.129,Y -502.879,Z 1336.902,A 0.000,B 0.000,C 90.000,E1 18.308} C_DIS
LIN {X 0.169,Y -494.922,Z 1336.897,A 0.000,B 0.000,C 90.000,E1 17.511} C_DIS
LIN {X -0.119,Y -486.393,Z 1336.893,A 0.000,B 0.000,C 90.000,E1 16.732} C_DIS
LIN {X 0.154,Y -473.487,Z 1336.886,A 0.000,B 0.000,C 90.000,E1 15.481} C_DIS
LIN {X -0.176,Y -457.629,Z 1336.878,A 0.000,B 0.000,C 90.000,E1 14.008} C_DIS
LIN {X -0.150,Y -437.447,Z 1336.867,A 0.000,B 0.000,C 90.000,E1 12.007} C_DIS
LIN {X -0.227,Y -420.417,Z 1336.857,A 0.000,B 0.000,C 90.000,E1 10.197} C_DIS
LIN {X 0.058,Y -406.266,Z 1336.848,A 0.000,B 0.000,C 90.000,E1 8.568} C_DIS
LIN {X 0.042,Y -399.286,Z 1336.843,A 0.000,B 0.000,C 90.000,E1 7.757} C_DIS
LIN {X -0.120,Y -395.878,Z 1336.841,A 0.000,B 0.000,C 90.000,E1 7.352} C_DIS
LIN {X -0.176,Y -394.979,Z 1336.840,A 0.000,B 0.000,C 90.000,E1 7.182} C_DIS
LIN {X 0.178,Y -394.977,Z 1336.840,A 0.000,B 0.000,C 90.000,E1 7.125} C_DIS
LIN {X -0.008,Y -395.016,Z 1336.840,A 0.000,B 0.000,C 90.000,E1 7.125} C_DIS
LIN {X -0.045,Y -395.027,Z 1336.840,A 0.000,B 0.000,C 90.000,E1 7.125} C_DIS
LIN {X 0.040,Y -395.996,Z 1336.839,A 0.000,B 0.000,C 90.000,E1 7.004} C_DIS
LIN {X -0.147,Y -400.239,Z 1336.837,A 0.000,B 0.000,C 90.000,E1 6.663} C_DIS
LIN {X 0.040,Y -415.145,Z 1336.831,A 0.000,B 0.000,C 90.000,E1 5.625} C_DIS
LIN {X 0.035,Y -419.888,Z 1336.829,A 0.000,B 0.000,C 90.000,E1 5.277} C_DIS
LIN {X -0.170,Y -424.541,Z 1336.827,A 0.000,B 0.000,C 90.000,E1 4.935} C_DIS
LIN {X 0.135,Y -430.594,Z 1336.824,A 0.000,B 0.000,C 90.000,E1 4.359} C_DIS
LIN {X 0.196,Y -436.437,Z 1336.821,A 0.000,B 0.000,C 90.000,E1 3.784} C_DIS
LIN {X -0.092,Y -443.641,Z 1336.817,A 0.000,B 0.000,C 90.000,E1 3.094} C_DIS
LIN {X 0.153,Y -449.124,Z 1336.814,A 0.000,B 0.000,C 90.000,E1 2.465} C_DIS
LIN {X -0.017,Y -455.877,Z 1336.810,A 0.000,B 0.000,C 90.000,E1 1.718} C_DIS
LIN {X -0.158,Y -462.163,Z 1336.805,A 0.000,B 0.000,C 90.000,E1 0.974} C_DIS
LIN {X -0.089,Y -468.185,Z 1336.801,A 0.000,B 0.000,C 90.000,E1 0.172} C_DIS
LIN {X 0.076,Y -474.032,Z 1336.796,A 0.000,B 0.000,C 90.000,E1 359.312} C_DIS
LIN {X -0.218,Y -479.013,Z 1336.792,A 0.000,B 0.000,C 90.000,E1 358.568} C_DIS
LIN {X 0.029,Y -483.628,Z 1336.788,A 0.000,B 0.000,C 90.000,E1 357.764} C_DIS
LIN {X 0.001,Y -488.743,Z 1336.782,A 0.000,B 0.000,C 90.000,E1 356.846} C_DIS
LIN {X -0.006,Y -491.196,Z 1336.780,A 0.000,B 0.000,C 90.000,E1 356.388} C_DIS
LIN {X -0.123,Y -494.852,Z 1336.776,A 0.000,B 0.000,C 90.000,E1 355.641} C_DIS
LIN {X -0.030,Y -498.899,Z 1336.771,A 0.000,B 0.000,C 90.000,E1 354.723} C_DIS
LIN {X 0.155,Y -502.686,Z 1336.766,A 0.000,B 0.000,C 90.000,E1 353.799} C_DIS
LIN {X 0.137,Y -505.548,Z 1336.762,A 0.000,B 0.000,C 90.000,E1 353.053} C_DIS
LIN {X -0.161,Y -509.606,Z 1336.755,A 0.000,B 0.000,C 90.000,E1 351.894} C_DIS
LIN {X -0.208,Y -510.630,Z 1336.753,A 0.000,B 0.000,C 90.000,E1 351.602} C_DIS
LIN {X 0.106,Y -513.156,Z 1336.748,A 0.000,B 0.000,C 90.000,E1 350.679} C_DIS
LIN {X 0.004,Y -516.204,Z 1336.742,A 0.000,B 0.000,C 90.000,E1 349.511} C_DIS
LIN {X -0.049,Y -518.811,Z 1336.735,A 0.000,B 0.000,C 90.000,E1 348.342} C_DIS
LIN {X -0.063,Y -520.554,Z 1336.730,A 0.000,B 0.000,C 90.000,E1 347.465} C_DIS
LIN {X -0.063,Y -522.504,Z 1336.724,A 0.000,B 0.000,C 90.000,E1 346.297} C_DIS
LIN {X 0.076,Y -523.739,Z 1336.719,A 0.000,B 0.000,C 90.000,E1 345.408} C_DIS
LIN {X -0.275,Y -524.684,Z 1336.714,A 0.000,B 0.000,C 90.000,E1 344.574} C_DIS
LIN {X -0.110,Y -525.360,Z 1336.709,A 0.000,B 0.000,C 90.000,E1 343.685} C_DIS
LIN {X 0.213,Y -525.910,Z 1336.704,A 0.000,B 0.000,C 90.000,E1 342.779} C_DIS
LIN {X -0.117,Y -526.125,Z 1336.700,A 0.000,B 0.000,C 90.000,E1 341.945} C_DIS
LIN {X -0.113,Y -525.956,Z 1336.693,A 0.000,B 0.000,C 90.000,E1 340.786} C_DIS
LIN {X 0.050,Y -525.686,Z 1336.690,A 0.000,B 0.000,C 90.000,E1 340.188} C_DIS
LIN {X -0.104,Y -525.317,Z 1336.687,A 0.000,B 0.000,C 90.000,E1 339.625} C_DIS
LIN {X 0.214,Y -524.291,Z 1336.682,A 0.000,B 0.000,C 90.000,E1 338.720} C_DIS
LIN {X 0.057,Y -523.502,Z 1336.679,A 0.000,B 0.000,C 90.000,E1 338.156} C_DIS
LIN {X 0.059,Y -522.052,Z 1336.674,A 0.000,B 0.000,C 90.000,E1 337.283} C_DIS
LIN {X 0.048,Y -520.366,Z 1336.669,A 0.000,B 0.000,C 90.000,E1 336.410} C_DIS
LIN {X -0.129,Y -519.100,Z 1336.666,A 0.000,B 0.000,C 90.000,E1 335.845} C_DIS
LIN {X -0.042,Y -516.024,Z 1336.659,A 0.000,B 0.000,C 90.000,E1 334.665} C_DIS
LIN {X -0.029,Y -514.226,Z 1336.656,A 0.000,B 0.000,C 90.000,E1 334.076} C_DIS
LIN {X 0.092,Y -513.147,Z 1336.654,A 0.000,B 0.000,C 90.000,E1 333.768} C_DIS
LIN {X 0.032,Y -511.245,Z 1336.652,A 0.000,B 0.000,C 90.000,E1 333.332} C_DIS
LIN {X 0.192,Y -508.940,Z 1336.649,A 0.000,B 0.000,C 90.000,E1 332.871} C_DIS
LIN {X -0.166,Y -506.925,Z 1336.648,A 0.000,B 0.000,C 90.000,E1 332.615} C_DIS
LIN {X 0.102,Y -505.505,Z 1336.647,A 0.000,B 0.000,C 90.000,E1 332.436} C_DIS
LIN {X 0.032,Y -496.490,Z 1336.644,A 0.000,B 0.000,C 90.000,E1 331.897} C_DIS
LIN {X 0.007,Y -470.921,Z 1336.635,A 0.000,B 0.000,C 90.000,E1 330.255} C_DIS
LIN {X 0.098,Y -447.351,Z 1336.625,A 0.000,B 0.000,C 90.000,E1 328.535} C_DIS
LIN {X 0.015,Y -425.771,Z 1336.616,A 0.000,B 0.000,C 90.000,E1 326.786} C_DIS
LIN {X -0.002,Y -404.652,Z 1336.605,A 0.000,B 0.000,C 90.000,E1 324.848} C_DIS
LIN {X 0.133,Y -385.521,Z 1336.594,A 0.000,B 0.000,C 90.000,E1 322.844} C_DIS
LIN {X -0.196,Y -373.690,Z 1336.586,A 0.000,B 0.000,C 90.000,E1 321.537} C_DIS
LIN {X -0.231,Y -373.673,Z 1336.586,A 0.000,B 0.000,C 90.000,E1 321.537} C_DIS
LIN {X -0.032,Y -378.003,Z 1336.564,A 0.000,B 0.000,C 90.000,E1 317.553} C_DIS
LIN {X 0.007,Y -379.380,Z 1336.554,A 0.000,B 0.000,C 90.000,E1 315.729} C_DIS
LIN {X 0.027,Y -384.611,Z 1336.528,A 0.000,B 0.000,C 90.000,E1 311.024} C_DIS
LIN {X 0.079,Y -385.218,Z 1336.524,A 0.000,B 0.000,C 90.000,E1 310.297} C_DIS
LIN {X -0.204,Y -391.270,Z 1336.492,A 0.000,B 0.000,C 90.000,E1 304.612} C_DIS
LIN {X -0.051,Y -396.983,Z 1336.459,A 0.000,B 0.000,C 90.000,E1 298.565} C_DIS
LIN {X -0.100,Y -401.348,Z 1336.427,A 0.000,B 0.000,C 90.000,E1 292.950} C_DIS
LIN {X -0.019,Y -401.657,Z 1336.426,A 0.000,B 0.000,C 90.000,E1 292.589} C_DIS
LIN {X 0.132,Y -404.748,Z 1336.395,A 0.000,B 0.000,C 90.000,E1 286.985} C_DIS
LIN {X 0.146,Y -406.156,Z 1336.364,A 0.000,B 0.000,C 90.000,E1 281.422} C_DIS
LIN {X -0.153,Y -405.676,Z 1336.333,A 0.000,B 0.000,C 90.000,E1 275.910} C_DIS
LIN {X -0.082,Y -403.565,Z 1336.306,A 0.000,B 0.000,C 90.000,E1 271.031} C_DIS
LIN {X -0.147,Y -403.175,Z 1336.302,A 0.000,B 0.000,C 90.000,E1 270.344} C_DIS
LIN {X 0.087,Y -399.064,Z 1336.273,A 0.000,B 0.000,C 90.000,E1 265.065} C_DIS
LIN {X 0.028,Y -398.769,Z 1336.271,A 0.000,B 0.000,C 90.000,E1 264.723} C_DIS
LIN {X -0.082,Y -393.288,Z 1336.243,A 0.000,B 0.000,C 90.000,E1 259.803} C_DIS
LIN {X -0.161,Y -392.663,Z 1336.239,A 0.000,B 0.000,C 90.000,E1 259.106} C_DIS
LIN {X 0.010,Y -386.242,Z 1336.214,A 0.000,B 0.000,C 90.000,E1 254.448} C_DIS
LIN {X -0.024,Y -385.145,Z 1336.208,A 0.000,B 0.000,C 90.000,E1 253.378} C_DIS
LIN {X 0.084,Y -377.810,Z 1336.182,A 0.000,B 0.000,C 90.000,E1 248.666} C_DIS
LIN {X -0.045,Y -376.078,Z 1336.173,A 0.000,B 0.000,C 90.000,E1 247.230} C_DIS
LIN {X 0.012,Y -368.746,Z 1336.149,A 0.000,B 0.000,C 90.000,E1 242.820} C_DIS
LIN {X -0.003,Y -366.393,Z 1336.139,A 0.000,B 0.000,C 90.000,E1 240.973} C_DIS
LIN {X 0.163,Y -365.093,Z 1336.135,A 0.000,B 0.000,C 90.000,E1 240.205} C_DIS
LIN {X -0.088,Y -358.497,Z 1336.112,A 0.000,B 0.000,C 90.000,E1 236.135} C_DIS
LIN {X -0.028,Y -356.173,Z 1336.101,A 0.000,B 0.000,C 90.000,E1 234.242} C_DIS
LIN {X -0.088,Y -354.923,Z 1336.097,A 0.000,B 0.000,C 90.000,E1 233.497} C_DIS
LIN {X -0.105,Y -348.153,Z 1336.072,A 0.000,B 0.000,C 90.000,E1 228.933} C_DIS
LIN {X 0.066,Y -346.050,Z 1336.061,A 0.000,B 0.000,C 90.000,E1 226.986} C_DIS
LIN {X 0.086,Y -340.791,Z 1336.041,A 0.000,B 0.000,C 90.000,E1 223.299} C_DIS
LIN {X 0.068,Y -340.803,Z 1336.041,A 0.000,B 0.000,C 90.000,E1 223.299} C_DIS
LIN {X -0.026,Y -356.677,Z 1336.028,A 0.000,B 0.000,C 90.000,E1 221.024} C_DIS
LIN {X -0.003,Y -373.865,Z 1336.016,A 0.000,B 0.000,C 90.000,E1 218.830} C_DIS
LIN {X 0.028,Y -391.571,Z 1336.005,A 0.000,B 0.000,C 90.000,E1 216.824} C_DIS
LIN {X 0.242,Y -411.255,Z 1335.994,A 0.000,B 0.000,C 90.000,E1 214.818} C_DIS
LIN {X -0.266,Y -432.947,Z 1335.983,A 0.000,B 0.000,C 90.000,E1 212.959} C_DIS
LIN {X 0.190,Y -443.958,Z 1335.978,A 0.000,B 0.000,C 90.000,E1 212.005} C_DIS
LIN {X -0.165,Y -445.277,Z 1335.977,A 0.000,B 0.000,C 90.000,E1 211.926} C_DIS
LIN {X 0.246,Y -446.945,Z 1335.976,A 0.000,B 0.000,C 90.000,E1 211.592} C_DIS
LIN {X 0.077,Y -448.255,Z 1335.974,A 0.000,B 0.000,C 90.000,E1 211.288} C_DIS
LIN {X -0.233,Y -449.272,Z 1335.972,A 0.000,B 0.000,C 90.000,E1 211.003} C_DIS
LIN {X -0.077,Y -450.832,Z 1335.969,A 0.000,B 0.000,C 90.000,E1 210.335} C_DIS
LIN {X 0.090,Y -451.948,Z 1335.965,A 0.000,B 0.000,C 90.000,E1 209.667} C_DIS
LIN {X 0.230,Y -453.484,Z 1335.958,A 0.000,B 0.000,C 90.000,E1 208.359} C_DIS
LIN {X 0.166,Y -456.856,Z 1335.943,A 0.000,B 0.000,C 90.000,E1 205.796} C_DIS
LIN {X 0.171,Y -458.651,Z 1335.936,A 0.000,B 0.000,C 90.000,E1 204.515} C_DIS
LIN {X 0.005,Y -460.375,Z 1335.929,A 0.000,B 0.000,C 90.000,E1 203.259} C_DIS
LIN {X 0.038,Y -462.428,Z 1335.920,A 0.000,B 0.000,C 90.000,E1 201.663} C_DIS
LIN {X -0.179,Y -463.747,Z 1335.915,A 0.000,B 0.000,C 90.000,E1 200.737} C_DIS
LIN {X -0.149,Y -466.017,Z 1335.905,A 0.000,B 0.000,C 90.000,E1 198.833} C_DIS
LIN {X 0.130,Y -467.939,Z 1335.896,A 0.000,B 0.000,C 90.000,E1 197.221} C_DIS
LIN {X 0.004,Y -469.677,Z 1335.887,A 0.000,B 0.000,C 90.000,E1 195.662} C_DIS
LIN {X -0.040,Y -470.996,Z 1335.880,A 0.000,B 0.000,C 90.000,E1 194.411} C_DIS
LIN {X -0.183,Y -472.419,Z 1335.873,A 0.000,B 0.000,C 90.000,E1 193.175} C_DIS
LIN {X 0.120,Y -474.836,Z 1335.861,A 0.000,B 0.000,C 90.000,E1 190.950} C_DIS
LIN {X 0.008,Y -476.865,Z 1335.851,A 0.000,B 0.000,C 90.000,E1 189.095} C_DIS
LIN {X -0.152,Y -478.119,Z 1335.844,A 0.000,B 0.000,C 90.000,E1 187.871} C_DIS
LIN {X -0.107,Y -479.533,Z 1335.835,A 0.000,B 0.000,C 90.000,E1 186.315} C_DIS
LIN {X 0.124,Y -480.419,Z 1335.828,A 0.000,B 0.000,C 90.000,E1 185.049} C_DIS
LIN {X -0.113,Y -481.130,Z 1335.821,A 0.000,B 0.000,C 90.000,E1 183.841} C_DIS
LIN {X 0.108,Y -481.636,Z 1335.814,A 0.000,B 0.000,C 90.000,E1 182.579} C_DIS
LIN {X -0.147,Y -481.807,Z 1335.808,A 0.000,B 0.000,C 90.000,E1 181.375} C_DIS
LIN {X -0.225,Y -481.852,Z 1335.802,A 0.000,B 0.000,C 90.000,E1 180.458} C_DIS
LIN {X -0.192,Y -481.425,Z 1335.794,A 0.000,B 0.000,C 90.000,E1 178.912} C_DIS
LIN {X 0.032,Y -480.844,Z 1335.787,A 0.000,B 0.000,C 90.000,E1 177.650} C_DIS
LIN {X -0.039,Y -480.178,Z 1335.782,A 0.000,B 0.000,C 90.000,E1 176.731} C_DIS
LIN {X -0.114,Y -479.210,Z 1335.777,A 0.000,B 0.000,C 90.000,E1 175.812} C_DIS
LIN {X -0.204,Y -478.072,Z 1335.772,A 0.000,B 0.000,C 90.000,E1 174.894} C_DIS
LIN {X -0.099,Y -477.212,Z 1335.768,A 0.000,B 0.000,C 90.000,E1 174.261} C_DIS
LIN {X -0.002,Y -476.091,Z 1335.765,A 0.000,B 0.000,C 90.000,E1 173.628} C_DIS
LIN {X -0.083,Y -474.118,Z 1335.760,A 0.000,B 0.000,C 90.000,E1 172.704} C_DIS
LIN {X 0.051,Y -472.509,Z 1335.756,A 0.000,B 0.000,C 90.000,E1 172.064} C_DIS
LIN {X 0.106,Y -470.461,Z 1335.753,A 0.000,B 0.000,C 90.000,E1 171.432} C_DIS
LIN {X 0.033,Y -466.897,Z 1335.747,A 0.000,B 0.000,C 90.000,E1 170.500} C_DIS
LIN {X -0.083,Y -461.998,Z 1335.742,A 0.000,B 0.000,C 90.000,E1 169.567} C_DIS
LIN {X 0.194,Y -456.361,Z 1335.737,A 0.000,B 0.000,C 90.000,E1 168.578} C_DIS
LIN {X -0.147,Y -446.969,Z 1335.729,A 0.000,B 0.000,C 90.000,E1 167.173} C_DIS
LIN {X -0.238,Y -438.541,Z 1335.721,A 0.000,B 0.000,C 90.000,E1 165.880} C_DIS
LIN {X 0.174,Y -428.956,Z 1335.713,A 0.000,B 0.000,C 90.000,E1 164.338} C_DIS
LIN {X 0.057,Y -424.829,Z 1335.709,A 0.000,B 0.000,C 90.000,E1 163.685} C_DIS
LIN {X -0.156,Y -423.065,Z 1335.708,A 0.000,B 0.000,C 90.000,E1 163.378} C_DIS
LIN {X 0.030,Y -421.690,Z 1335.706,A 0.000,B 0.000,C 90.000,E1 163.015} C_DIS
LIN {X 0.085,Y -420.611,Z 1335.704,A 0.000,B 0.000,C 90.000,E1 162.670} C_DIS
LIN {X -0.131,Y -419.907,Z 1335.702,A 0.000,B 0.000,C 90.000,E1 162.308} C_DIS
LIN {X 0.005,Y -419.891,Z 1335.701,A 0.000,B 0.000,C 90.000,E1 162.236} C_DIS
LIN {X 0.014,Y -420.898,Z 1335.699,A 0.000,B 0.000,C 90.000,E1 161.873} C_DIS
LIN {X -0.015,Y -421.008,Z 1335.699,A 0.000,B 0.000,C 90.000,E1 161.819} C_DIS
LIN {X -0.054,Y -421.047,Z 1335.699,A 0.000,B 0.000,C 90.000,E1 161.819} C_DIS
LIN {X -0.035,Y -423.508,Z 1335.697,A 0.000,B 0.000,C 90.000,E1 161.456} C_DIS
LIN {X 0.056,Y -425.134,Z 1335.696,A 0.000,B 0.000,C 90.000,E1 161.275} C_DIS
LIN {X -0.169,Y -429.774,Z 1335.694,A 0.000,B 0.000,C 90.000,E1 160.859} C_DIS
LIN {X -0.195,Y -434.981,Z 1335.691,A 0.000,B 0.000,C 90.000,E1 160.423} C_DIS
LIN {X 0.066,Y -447.322,Z 1335.686,A 0.000,B 0.000,C 90.000,E1 159.444} C_DIS
LIN {X 0.184,Y -459.811,Z 1335.681,A 0.000,B 0.000,C 90.000,E1 158.465} C_DIS
LIN {X -0.224,Y -469.114,Z 1335.677,A 0.000,B 0.000,C 90.000,E1 157.794} C_DIS
LIN {X -0.222,Y -479.762,Z 1335.672,A 0.000,B 0.000,C 90.000,E1 156.922} C_DIS
LIN {X 0.199,Y -487.041,Z 1335.668,A 0.000,B 0.000,C 90.000,E1 156.230} C_DIS
LIN {X -0.226,Y -494.130,Z 1335.664,A 0.000,B 0.000,C 90.000,E1 155.613} C_DIS
LIN {X -0.091,Y -499.684,Z 1335.661,A 0.000,B 0.000,C 90.000,E1 155.049} C_DIS
LIN {X 0.025,Y -506.494,Z 1335.657,A 0.000,B 0.000,C 90.000,E1 154.332} C_DIS
LIN {X -0.122,Y -512.824,Z 1335.654,A 0.000,B 0.000,C 90.000,E1 153.640} C_DIS
LIN {X -0.010,Y -517.685,Z 1335.650,A 0.000,B 0.000,C 90.000,E1 153.050} C_DIS
LIN {X -0.050,Y -521.157,Z 1335.648,A 0.000,B 0.000,C 90.000,E1 152.615} C_DIS
LIN {X 0.007,Y -525.330,Z 1335.645,A 0.000,B 0.000,C 90.000,E1 152.025} C_DIS
LIN {X 0.096,Y -528.969,Z 1335.641,A 0.000,B 0.000,C 90.000,E1 151.435} C_DIS
LIN {X 0.066,Y -532.693,Z 1335.637,A 0.000,B 0.000,C 90.000,E1 150.717} C_DIS
LIN {X 0.064,Y -535.623,Z 1335.633,A 0.000,B 0.000,C 90.000,E1 149.999} C_DIS
LIN {X 0.225,Y -537.651,Z 1335.630,A 0.000,B 0.000,C 90.000,E1 149.410} C_DIS
LIN {X -0.061,Y -540.151,Z 1335.625,A 0.000,B 0.000,C 90.000,E1 148.584} C_DIS
LIN {X 0.132,Y -541.691,Z 1335.622,A 0.000,B 0.000,C 90.000,E1 147.995} C_DIS
LIN {X -0.127,Y -543.064,Z 1335.619,A 0.000,B 0.000,C 90.000,E1 147.454} C_DIS
LIN {X 0.104,Y -544.779,Z 1335.615,A 0.000,B 0.000,C 90.000,E1 146.580} C_DIS
LIN {X -0.104,Y -546.267,Z 1335.610,A 0.000,B 0.000,C 90.000,E1 145.754} C_DIS
LIN {X 0.016,Y -547.429,Z 1335.605,A 0.000,B 0.000,C 90.000,E1 144.895} C_DIS
LIN {X -0.165,Y -548.372,Z 1335.600,A 0.000,B 0.000,C 90.000,E1 144.069} C_DIS
LIN {X 0.035,Y -549.347,Z 1335.594,A 0.000,B 0.000,C 90.000,E1 142.924} C_DIS
LIN {X 0.032,Y -550.771,Z 1335.582,A 0.000,B 0.000,C 90.000,E1 140.678} C_DIS
LIN {X -0.070,Y -552.346,Z 1335.569,A 0.000,B 0.000,C 90.000,E1 138.447} C_DIS
LIN {X 0.038,Y -553.148,Z 1335.566,A 0.000,B 0.000,C 90.000,E1 137.877} C_DIS
LIN {X 0.055,Y -553.451,Z 1335.564,A 0.000,B 0.000,C 90.000,E1 137.595} C_DIS
LIN {X -0.051,Y -554.421,Z 1335.562,A 0.000,B 0.000,C 90.000,E1 137.187} C_DIS
LIN {X 0.042,Y -554.732,Z 1335.561,A 0.000,B 0.000,C 90.000,E1 137.025} C_DIS
LIN {X 0.000,Y -554.769,Z 1335.561,A 0.000,B 0.000,C 90.000,E1 137.025} C_DIS
LIN {X -0.112,Y -555.547,Z 1335.561,A 0.000,B 0.000,C 90.000,E1 136.986} C_DIS
LIN {X 0.099,Y -557.547,Z 1335.560,A 0.000,B 0.000,C 90.000,E1 136.863} C_DIS
LIN {X -0.052,Y -568.355,Z 1335.559,A 0.000,B 0.000,C 90.000,E1 136.581} C_DIS
LIN {X -0.231,Y -574.900,Z 1335.558,A 0.000,B 0.000,C 90.000,E1 136.377} C_DIS
LIN {X 0.208,Y -577.788,Z 1335.557,A 0.000,B 0.000,C 90.000,E1 136.215} C_DIS
LIN {X 0.284,Y -583.350,Z 1335.555,A 0.000,B 0.000,C 90.000,E1 135.891} C_DIS
LIN {X 0.041,Y -586.313,Z 1335.554,A 0.000,B 0.000,C 90.000,E1 135.729} C_DIS
LIN {X 0.033,Y -591.969,Z 1335.552,A 0.000,B 0.000,C 90.000,E1 135.324} C_DIS
LIN {X 0.142,Y -598.662,Z 1335.549,A 0.000,B 0.000,C 90.000,E1 134.757} C_DIS
LIN {X 0.263,Y -601.431,Z 1335.547,A 0.000,B 0.000,C 90.000,E1 134.514} C_DIS
LIN {X 0.226,Y -606.470,Z 1335.545,A 0.000,B 0.000,C 90.000,E1 134.028} C_DIS
LIN {X -0.047,Y -610.995,Z 1335.542,A 0.000,B 0.000,C 90.000,E1 133.581} C_DIS
LIN {X 0.056,Y -615.639,Z 1335.539,A 0.000,B 0.000,C 90.000,E1 133.056} C_DIS
LIN {X 0.026,Y -622.068,Z 1335.535,A 0.000,B 0.000,C 90.000,E1 132.285} C_DIS
LIN {X 0.197,Y -626.096,Z 1335.532,A 0.000,B 0.000,C 90.000,E1 131.757} C_DIS
LIN {X 0.073,Y -630.814,Z 1335.529,A 0.000,B 0.000,C 90.000,E1 131.148} C_DIS
LIN {X 0.179,Y -637.220,Z 1335.524,A 0.000,B 0.000,C 90.000,E1 130.253} C_DIS
LIN {X 0.027,Y -643.315,Z 1335.519,A 0.000,B 0.000,C 90.000,E1 129.402} C_DIS
LIN {X 0.061,Y -649.827,Z 1335.514,A 0.000,B 0.000,C 90.000,E1 128.418} C_DIS
LIN {X -0.039,Y -654.536,Z 1335.509,A 0.000,B 0.000,C 90.000,E1 127.684} C_DIS
LIN {X -0.130,Y -658.342,Z 1335.506,A 0.000,B 0.000,C 90.000,E1 127.076} C_DIS
LIN {X -0.014,Y -664.591,Z 1335.500,A 0.000,B 0.000,C 90.000,E1 125.964} C_DIS
LIN {X 0.055,Y -667.046,Z 1335.497,A 0.000,B 0.000,C 90.000,E1 125.471} C_DIS
LIN {X 0.099,Y -670.460,Z 1335.493,A 0.000,B 0.000,C 90.000,E1 124.739} C_DIS
LIN {X -0.214,Y -673.518,Z 1335.489,A 0.000,B 0.000,C 90.000,E1 124.040} C_DIS
LIN {X -0.098,Y -675.314,Z 1335.486,A 0.000,B 0.000,C 90.000,E1 123.547} C_DIS
LIN {X -0.173,Y -677.634,Z 1335.482,A 0.000,B 0.000,C 90.000,E1 122.832} C_DIS
LIN {X 0.151,Y -679.701,Z 1335.478,A 0.000,B 0.000,C 90.000,E1 122.084} C_DIS
LIN {X -0.087,Y -681.522,Z 1335.474,A 0.000,B 0.000,C 90.000,E1 121.386} C_DIS
LIN {X -0.082,Y -683.086,Z 1335.470,A 0.000,B 0.000,C 90.000,E1 120.669} C_DIS
LIN {X -0.262,Y -684.023,Z 1335.468,A 0.000,B 0.000,C 90.000,E1 120.207} C_DIS
LIN {X 0.114,Y -685.115,Z 1335.464,A 0.000,B 0.000,C 90.000,E1 119.461} C_DIS
LIN {X 0.160,Y -685.883,Z 1335.460,A 0.000,B 0.000,C 90.000,E1 118.743} C_DIS
LIN {X 0.213,Y -686.334,Z 1335.456,A 0.000,B 0.000,C 90.000,E1 118.025} C_DIS
LIN {X 0.179,Y -686.539,Z 1335.451,A 0.000,B 0.000,C 90.000,E1 117.078} C_DIS
LIN {X 0.239,Y -686.493,Z 1335.447,A 0.000,B 0.000,C 90.000,E1 116.360} C_DIS
LIN {X -0.008,Y -686.144,Z 1335.443,A 0.000,B 0.000,C 90.000,E1 115.668} C_DIS
LIN {X -0.183,Y -685.742,Z 1335.440,A 0.000,B 0.000,C 90.000,E1 115.207} C_DIS
LIN {X -0.033,Y -685.127,Z 1335.437,A 0.000,B 0.000,C 90.000,E1 114.719} C_DIS
LIN {X -0.221,Y -684.072,Z 1335.435,A 0.000,B 0.000,C 90.000,E1 114.259} C_DIS
LIN {X -0.008,Y -683.294,Z 1335.433,A 0.000,B 0.000,C 90.000,E1 114.003} C_DIS
LIN {X 0.134,Y -681.169,Z 1335.431,A 0.000,B 0.000,C 90.000,E1 113.515} C_DIS
LIN {X 0.235,Y -680.350,Z 1335.430,A 0.000,B 0.000,C 90.000,E1 113.387} C_DIS
LIN {X -0.264,Y -675.928,Z 1335.427,A 0.000,B 0.000,C 90.000,E1 112.950} C_DIS
LIN {X -0.171,Y -674.411,Z 1335.427,A 0.000,B 0.000,C 90.000,E1 112.823} C_DIS
LIN {X 0.021,Y -668.702,Z 1335.425,A 0.000,B 0.000,C 90.000,E1 112.514} C_DIS
LIN {X -0.241,Y -665.306,Z 1335.424,A 0.000,B 0.000,C 90.000,E1 112.386} C_DIS
LIN {X 0.383,Y -661.015,Z 1335.424,A 0.000,B 0.000,C 90.000,E1 112.206} C_DIS
LIN {X -0.254,Y -658.960,Z 1335.423,A 0.000,B 0.000,C 90.000,E1 112.206} C_DIS
LIN {X 0.078,Y -649.662,Z 1335.422,A 0.000,B 0.000,C 90.000,E1 112.025} C_DIS
LIN {X 0.078,Y -646.049,Z 1335.422,A 0.000,B 0.000,C 90.000,E1 111.972} C_DIS
LIN {X -0.234,Y -640.931,Z 1335.422,A 0.000,B 0.000,C 90.000,E1 111.897} C_DIS
LIN {X -0.275,Y -640.815,Z 1335.422,A 0.000,B 0.000,C 90.000,E1 111.897} C_DIS
LIN {X -0.114,Y -642.710,Z 1335.420,A 0.000,B 0.000,C 90.000,E1 111.589} C_DIS
LIN {X -0.110,Y -647.171,Z 1335.417,A 0.000,B 0.000,C 90.000,E1 111.046} C_DIS
LIN {X -0.195,Y -651.039,Z 1335.414,A 0.000,B 0.000,C 90.000,E1 110.556} C_DIS
LIN {X -0.167,Y -655.928,Z 1335.410,A 0.000,B 0.000,C 90.000,E1 109.812} C_DIS
LIN {X -0.199,Y -658.767,Z 1335.407,A 0.000,B 0.000,C 90.000,E1 109.322} C_DIS
LIN {X 0.248,Y -661.769,Z 1335.404,A 0.000,B 0.000,C 90.000,E1 108.671} C_DIS
LIN {X 0.157,Y -664.964,Z 1335.400,A 0.000,B 0.000,C 90.000,E1 107.946} C_DIS
LIN {X 0.093,Y -667.776,Z 1335.396,A 0.000,B 0.000,C 90.000,E1 107.221} C_DIS
LIN {X 0.051,Y -670.310,Z 1335.392,A 0.000,B 0.000,C 90.000,E1 106.496} C_DIS
LIN {X -0.091,Y -671.797,Z 1335.389,A 0.000,B 0.000,C 90.000,E1 106.024} C_DIS
LIN {X -0.101,Y -673.699,Z 1335.385,A 0.000,B 0.000,C 90.000,E1 105.300} C_DIS
LIN {X -0.276,Y -675.318,Z 1335.381,A 0.000,B 0.000,C 90.000,E1 104.592} C_DIS
LIN {X 0.325,Y -675.821,Z 1335.380,A 0.000,B 0.000,C 90.000,E1 104.300} C_DIS
LIN {X 0.175,Y -676.882,Z 1335.376,A 0.000,B 0.000,C 90.000,E1 103.592} C_DIS
LIN {X 0.081,Y -677.423,Z 1335.373,A 0.000,B 0.000,C 90.000,E1 103.119} C_DIS
LIN {X -0.105,Y -677.752,Z 1335.368,A 0.000,B 0.000,C 90.000,E1 102.175} C_DIS
LIN {X 0.280,Y -677.645,Z 1335.364,A 0.000,B 0.000,C 90.000,E1 101.422} C_DIS
LIN {X 0.185,Y -677.234,Z 1335.361,A 0.000,B 0.000,C 90.000,E1 100.950} C_DIS
LIN {X -0.092,Y -676.261,Z 1335.357,A 0.000,B 0.000,C 90.000,E1 100.254} C_DIS
LIN {X -0.202,Y -675.342,Z 1335.354,A 0.000,B 0.000,C 90.000,E1 99.782} C_DIS
LIN {X 0.232,Y -674.191,Z 1335.352,A 0.000,B 0.000,C 90.000,E1 99.265} C_DIS
LIN {X -0.003,Y -672.638,Z 1335.349,A 0.000,B 0.000,C 90.000,E1 98.803} C_DIS
LIN {X -0.319,Y -669.815,Z 1335.345,A 0.000,B 0.000,C 90.000,E1 98.106} C_DIS
LIN {X 0.087,Y -667.674,Z 1335.342,A 0.000,B 0.000,C 90.000,E1 97.587} C_DIS
LIN {X -0.190,Y -664.747,Z 1335.339,A 0.000,B 0.000,C 90.000,E1 97.004} C_DIS
LIN {X -0.012,Y -660.936,Z 1335.335,A 0.000,B 0.000,C 90.000,E1 96.258} C_DIS
LIN {X 0.328,Y -658.123,Z 1335.332,A 0.000,B 0.000,C 90.000,E1 95.739} C_DIS
LIN {X 0.095,Y -655.837,Z 1335.330,A 0.000,B 0.000,C 90.000,E1 95.391} C_DIS
LIN {X -0.279,Y -652.685,Z 1335.327,A 0.000,B 0.000,C 90.000,E1 94.935} C_DIS
LIN {X -0.106,Y -648.313,Z 1335.324,A 0.000,B 0.000,C 90.000,E1 94.302} C_DIS
LIN {X 0.142,Y -644.634,Z 1335.321,A 0.000,B 0.000,C 90.000,E1 93.784} C_DIS
LIN {X -0.318,Y -640.615,Z 1335.318,A 0.000,B 0.000,C 90.000,E1 93.326} C_DIS
LIN {X -0.128,Y -636.140,Z 1335.316,A 0.000,B 0.000,C 90.000,E1 92.808} C_DIS
LIN {X 0.000,Y -629.975,Z 1335.312,A 0.000,B 0.000,C 90.000,E1 92.178} C_DIS
LIN {X -0.125,Y -618.591,Z 1335.306,A 0.000,B 0.000,C 90.000,E1 91.088} C_DIS
LIN {X -0.297,Y -614.405,Z 1335.304,A 0.000,B 0.000,C 90.000,E1 90.745} C_DIS
LIN {X -0.072,Y -609.060,Z 1335.302,A 0.000,B 0.000,C 90.000,E1 90.286} C_DIS
LIN {X -0.073,Y -602.589,Z 1335.299,A 0.000,B 0.000,C 90.000,E1 89.885} C_DIS
LIN {X -0.206,Y -595.508,Z 1335.297,A 0.000,B 0.000,C 90.000,E1 89.542} C_DIS
LIN {X 0.178,Y -588.342,Z 1335.296,A 0.000,B 0.000,C 90.000,E1 89.198} C_DIS
LIN {X 0.269,Y -581.408,Z 1335.294,A 0.000,B 0.000,C 90.000,E1 88.912} C_DIS
LIN {X -0.019,Y -577.143,Z 1335.293,A 0.000,B 0.000,C 90.000,E1 88.740} C_DIS
LIN {X 0.204,Y -574.428,Z 1335.292,A 0.000,B 0.000,C 90.000,E1 88.511} C_DIS
LIN {X 0.189,Y -573.132,Z 1335.291,A 0.000,B 0.000,C 90.000,E1 88.396} C_DIS
LIN {X 0.155,Y -573.112,Z 1335.291,A 0.000,B 0.000,C 90.000,E1 88.396} C_DIS
LIN {X 0.048,Y -572.505,Z 1335.290,A 0.000,B 0.000,C 90.000,E1 88.165} C_DIS
LIN {X 0.125,Y -572.344,Z 1335.288,A 0.000,B 0.000,C 90.000,E1 87.879} C_DIS
LIN {X 0.264,Y -572.350,Z 1335.287,A 0.000,B 0.000,C 90.000,E1 87.593} C_DIS
LIN {X 0.027,Y -574.872,Z 1335.272,A 0.000,B 0.000,C 90.000,E1 84.894} C_DIS
LIN {X -0.156,Y -577.696,Z 1335.258,A 0.000,B 0.000,C 90.000,E1 82.470} C_DIS
LIN {X 0.178,Y -579.337,Z 1335.251,A 0.000,B 0.000,C 90.000,E1 81.084} C_DIS
LIN {X 0.052,Y -580.965,Z 1335.243,A 0.000,B 0.000,C 90.000,E1 79.746} C_DIS
LIN {X -0.051,Y -582.367,Z 1335.236,A 0.000,B 0.000,C 90.000,E1 78.409} C_DIS
LIN {X -0.019,Y -583.657,Z 1335.228,A 0.000,B 0.000,C 90.000,E1 77.061} C_DIS
LIN {X 0.172,Y -584.767,Z 1335.221,A 0.000,B 0.000,C 90.000,E1 75.700} C_DIS
LIN {X 0.060,Y -585.858,Z 1335.212,A 0.000,B 0.000,C 90.000,E1 74.102} C_DIS
LIN {X 0.215,Y -586.640,Z 1335.206,A 0.000,B 0.000,C 90.000,E1 73.015} C_DIS
LIN {X -0.168,Y -587.996,Z 1335.194,A 0.000,B 0.000,C 90.000,E1 70.913} C_DIS
LIN {X 0.320,Y -588.961,Z 1335.185,A 0.000,B 0.000,C 90.000,E1 69.263} C_DIS
LIN {X -0.156,Y -589.830,Z 1335.178,A 0.000,B 0.000,C 90.000,E1 67.975} C_DIS
LIN {X -0.066,Y -591.085,Z 1335.167,A 0.000,B 0.000,C 90.000,E1 66.102} C_DIS
LIN {X -0.288,Y -592.045,Z 1335.160,A 0.000,B 0.000,C 90.000,E1 64.793} C_DIS
LIN {X -0.083,Y -593.202,Z 1335.151,A 0.000,B 0.000,C 90.000,E1 63.179} C_DIS
LIN {X -0.119,Y -595.135,Z 1335.138,A 0.000,B 0.000,C 90.000,E1 60.795} C_DIS
LIN {X 0.046,Y -597.202,Z 1335.126,A 0.000,B 0.000,C 90.000,E1 58.663} C_DIS
LIN {X -0.058,Y -598.843,Z 1335.117,A 0.000,B 0.000,C 90.000,E1 57.089} C_DIS
LIN {X -0.126,Y -600.461,Z 1335.108,A 0.000,B 0.000,C 90.000,E1 55.515} C_DIS
LIN {X -0.079,Y -601.787,Z 1335.101,A 0.000,B 0.000,C 90.000,E1 54.196} C_DIS
LIN {X -0.252,Y -603.250,Z 1335.092,A 0.000,B 0.000,C 90.000,E1 52.637} C_DIS
LIN {X 0.083,Y -604.164,Z 1335.085,A 0.000,B 0.000,C 90.000,E1 51.295} C_DIS
LIN {X -0.200,Y -604.919,Z 1335.079,A 0.000,B 0.000,C 90.000,E1 50.275} C_DIS
LIN {X -0.088,Y -605.490,Z 1335.073,A 0.000,B 0.000,C 90.000,E1 49.218} C_DIS
LIN {X 0.030,Y -605.864,Z 1335.068,A 0.000,B 0.000,C 90.000,E1 48.162} C_DIS
LIN {X -0.107,Y -606.016,Z 1335.063,A 0.000,B 0.000,C 90.000,E1 47.391} C_DIS
LIN {X 0.036,Y -606.239,Z 1335.055,A 0.000,B 0.000,C 90.000,E1 45.810} C_DIS
LIN {X 0.131,Y -606.222,Z 1335.049,A 0.000,B 0.000,C 90.000,E1 44.757} C_DIS
LIN {X 0.223,Y -606.006,Z 1335.043,A 0.000,B 0.000,C 90.000,E1 43.704} C_DIS
LIN {X -0.050,Y -605.430,Z 1335.034,A 0.000,B 0.000,C 90.000,E1 42.162} C_DIS
LIN {X -0.388,Y -605.045,Z 1335.028,A 0.000,B 0.000,C 90.000,E1 41.148} C_DIS
LIN {X 0.031,Y -604.143,Z 1335.018,A 0.000,B 0.000,C 90.000,E1 39.277} C_DIS
LIN {X 0.120,Y -603.625,Z 1335.012,A 0.000,B 0.000,C 90.000,E1 38.222} C_DIS
LIN {X -0.289,Y -602.587,Z 1335.005,A 0.000,B 0.000,C 90.000,E1 36.950} C_DIS
LIN {X -0.115,Y -601.201,Z 1334.999,A 0.000,B 0.000,C 90.000,E1 35.884} C_DIS
LIN {X -0.208,Y -599.957,Z 1334.995,A 0.000,B 0.000,C 90.000,E1 35.105} C_DIS
LIN {X 0.178,Y -598.583,Z 1334.991,A 0.000,B 0.000,C 90.000,E1 34.278} C_DIS
LIN {X 0.052,Y -597.019,Z 1334.986,A 0.000,B 0.000,C 90.000,E1 33.499} C_DIS
LIN {X 0.080,Y -595.258,Z 1334.982,A 0.000,B 0.000,C 90.000,E1 32.704} C_DIS
LIN {X -0.090,Y -593.261,Z 1334.977,A 0.000,B 0.000,C 90.000,E1 31.926} C_DIS
LIN {X 0.011,Y -591.732,Z 1334.974,A 0.000,B 0.000,C 90.000,E1 31.386} C_DIS
LIN {X -0.009,Y -589.219,Z 1334.970,A 0.000,B 0.000,C 90.000,E1 30.590} C_DIS
LIN {X -0.055,Y -586.301,Z 1334.966,A 0.000,B 0.000,C 90.000,E1 29.795} C_DIS
LIN {X -0.292,Y -584.201,Z 1334.963,A 0.000,B 0.000,C 90.000,E1 29.283} C_DIS
LIN {X 0.123,Y -580.619,Z 1334.958,A 0.000,B 0.000,C 90.000,E1 28.437} C_DIS
LIN {X 0.127,Y -578.060,Z 1334.955,A 0.000,B 0.000,C 90.000,E1 27.897} C_DIS
LIN {X -0.239,Y -574.557,Z 1334.951,A 0.000,B 0.000,C 90.000,E1 27.257} C_DIS
LIN {X 0.056,Y -569.997,Z 1334.947,A 0.000,B 0.000,C 90.000,E1 26.411} C_DIS
LIN {X 0.136,Y -565.799,Z 1334.943,A 0.000,B 0.000,C 90.000,E1 25.720} C_DIS
LIN {X -0.233,Y -562.208,Z 1334.940,A 0.000,B 0.000,C 90.000,E1 25.207} C_DIS
LIN {X 0.175,Y -555.479,Z 1334.935,A 0.000,B 0.000,C 90.000,E1 24.207} C_DIS
LIN {X 0.225,Y -550.138,Z 1334.931,A 0.000,B 0.000,C 90.000,E1 23.515} C_DIS
LIN {X 0.252,Y -545.663,Z 1334.928,A 0.000,B 0.000,C 90.000,E1 22.950} C_DIS
LIN {X -0.126,Y -542.098,Z 1334.925,A 0.000,B 0.000,C 90.000,E1 22.567} C_DIS
LIN {X -0.147,Y -532.349,Z 1334.919,A 0.000,B 0.000,C 90.000,E1 21.461} C_DIS
LIN {X -0.230,Y -523.117,Z 1334.914,A 0.000,B 0.000,C 90.000,E1 20.482} C_DIS
LIN {X 0.263,Y -512.584,Z 1334.908,A 0.000,B 0.000,C 90.000,E1 19.322} C_DIS
LIN {X 0.039,Y -503.238,Z 1334.902,A 0.000,B 0.000,C 90.000,E1 18.362} C_DIS
LIN {X -0.026,Y -492.705,Z 1334.896,A 0.000,B 0.000,C 90.000,E1 17.330} C_DIS
LIN {X -0.077,Y -479.967,Z 1334.890,A 0.000,B 0.000,C 90.000,E1 16.134} C_DIS
LIN {X 0.196,Y -468.424,Z 1334.884,A 0.000,B 0.000,C 90.000,E1 15.009} C_DIS
LIN {X 0.137,Y -455.379,Z 1334.877,A 0.000,B 0.000,C 90.000,E1 13.772} C_DIS
LIN {X -0.183,Y -431.084,Z 1334.863,A 0.000,B 0.000,C 90.000,E1 11.366} C_DIS
LIN {X 0.196,Y -415.432,Z 1334.854,A 0.000,B 0.000,C 90.000,E1 9.613} C_DIS
LIN {X 0.118,Y -404.071,Z 1334.846,A 0.000,B 0.000,C 90.000,E1 8.341} C_DIS
LIN {X 0.096,Y -399.988,Z 1334.844,A 0.000,B 0.000,C 90.000,E1 7.871} C_DIS
LIN {X 0.006,Y -395.842,Z 1334.841,A 0.000,B 0.000,C 90.000,E1 7.352} C_DIS
LIN {X -0.149,Y -395.213,Z 1334.840,A 0.000,B 0.000,C 90.000,E1 7.239} C_DIS
LIN {X -0.183,Y -395.205,Z 1334.840,A 0.000,B 0.000,C 90.000,E1 7.239} C_DIS
LIN {X -0.034,Y -395.373,Z 1334.840,A 0.000,B 0.000,C 90.000,E1 7.125} C_DIS
LIN {X -0.072,Y -395.404,Z 1334.840,A 0.000,B 0.000,C 90.000,E1 7.125} C_DIS
LIN {X -0.086,Y -399.821,Z 1334.837,A 0.000,B 0.000,C 90.000,E1 6.720} C_DIS
LIN {X -0.179,Y -414.691,Z 1334.832,A 0.000,B 0.000,C 90.000,E1 5.739} C_DIS
LIN {X -0.124,Y -419.379,Z 1334.830,A 0.000,B 0.000,C 90.000,E1 5.391} C_DIS
LIN {X 0.150,Y -424.029,Z 1334.828,A 0.000,B 0.000,C 90.000,E1 4.992} C_DIS
LIN {X 0.156,Y -430.032,Z 1334.825,A 0.000,B 0.000,C 90.000,E1 4.473} C_DIS
LIN {X -0.100,Y -435.883,Z 1334.822,A 0.000,B 0.000,C 90.000,E1 3.955} C_DIS
LIN {X 0.054,Y -443.123,Z 1334.818,A 0.000,B 0.000,C 90.000,E1 3.212} C_DIS
LIN {X -0.063,Y -448.728,Z 1334.815,A 0.000,B 0.000,C 90.000,E1 2.636} C_DIS
LIN {X -0.203,Y -455.528,Z 1334.810,A 0.000,B 0.000,C 90.000,E1 1.892} C_DIS
LIN {X -0.102,Y -462.136,Z 1334.806,A 0.000,B 0.000,C 90.000,E1 1.088} C_DIS
LIN {X 0.222,Y -469.317,Z 1334.801,A 0.000,B 0.000,C 90.000,E1 0.115} C_DIS
LIN {X 0.082,Y -475.005,Z 1334.796,A 0.000,B 0.000,C 90.000,E1 359.312} C_DIS
LIN {X -0.203,Y -479.985,Z 1334.792,A 0.000,B 0.000,C 90.000,E1 358.568} C_DIS
LIN {X 0.054,Y -484.573,Z 1334.788,A 0.000,B 0.000,C 90.000,E1 357.764} C_DIS
LIN {X 0.037,Y -489.689,Z 1334.783,A 0.000,B 0.000,C 90.000,E1 356.846} C_DIS
LIN {X 0.034,Y -492.137,Z 1334.780,A 0.000,B 0.000,C 90.000,E1 356.388} C_DIS
LIN {X -0.073,Y -495.796,Z 1334.776,A 0.000,B 0.000,C 90.000,E1 355.641} C_DIS
LIN {X 0.031,Y -499.845,Z 1334.771,A 0.000,B 0.000,C 90.000,E1 354.723} C_DIS
LIN {X 0.229,Y -503.650,Z 1334.766,A 0.000,B 0.000,C 90.000,E1 353.799} C_DIS
LIN {X 0.219,Y -506.487,Z 1334.762,A 0.000,B 0.000,C 90.000,E1 353.053} C_DIS
LIN {X -0.107,Y -511.614,Z 1334.753,A 0.000,B 0.000,C 90.000,E1 351.602} C_DIS
LIN {X 0.217,Y -514.163,Z 1334.748,A 0.000,B 0.000,C 90.000,E1 350.679} C_DIS
LIN {X 0.132,Y -517.242,Z 1334.742,A 0.000,B 0.000,C 90.000,E1 349.511} C_DIS
LIN {X 0.095,Y -519.839,Z 1334.735,A 0.000,B 0.000,C 90.000,E1 348.342} C_DIS
LIN {X 0.092,Y -521.596,Z 1334.730,A 0.000,B 0.000,C 90.000,E1 347.465} C_DIS
LIN {X 0.108,Y -523.561,Z 1334.724,A 0.000,B 0.000,C 90.000,E1 346.297} C_DIS
LIN {X -0.249,Y -524.800,Z 1334.719,A 0.000,B 0.000,C 90.000,E1 345.463} C_DIS
LIN {X -0.080,Y -525.762,Z 1334.714,A 0.000,B 0.000,C 90.000,E1 344.574} C_DIS
LIN {X 0.086,Y -526.289,Z 1334.711,A 0.000,B 0.000,C 90.000,E1 343.976} C_DIS
LIN {X -0.071,Y -526.993,Z 1334.705,A 0.000,B 0.000,C 90.000,E1 342.834} C_DIS
LIN {X 0.115,Y -527.222,Z 1334.700,A 0.000,B 0.000,C 90.000,E1 341.945} C_DIS
LIN {X 0.134,Y -527.062,Z 1334.693,A 0.000,B 0.000,C 90.000,E1 340.786} C_DIS
LIN {X -0.190,Y -526.798,Z 1334.690,A 0.000,B 0.000,C 90.000,E1 340.242} C_DIS
LIN {X -0.024,Y -526.426,Z 1334.687,A 0.000,B 0.000,C 90.000,E1 339.645} C_DIS
LIN {X -0.172,Y -525.822,Z 1334.684,A 0.000,B 0.000,C 90.000,E1 339.082} C_DIS
LIN {X -0.147,Y -524.648,Z 1334.679,A 0.000,B 0.000,C 90.000,E1 338.209} C_DIS
LIN {X 0.153,Y -523.187,Z 1334.674,A 0.000,B 0.000,C 90.000,E1 337.305} C_DIS
LIN {X -0.169,Y -522.545,Z 1334.672,A 0.000,B 0.000,C 90.000,E1 337.050} C_DIS
LIN {X 0.146,Y -521.508,Z 1334.669,A 0.000,B 0.000,C 90.000,E1 336.433} C_DIS
LIN {X 0.334,Y -519.555,Z 1334.664,A 0.000,B 0.000,C 90.000,E1 335.537} C_DIS
LIN {X -0.181,Y -517.193,Z 1334.659,A 0.000,B 0.000,C 90.000,E1 334.717} C_DIS
LIN {X -0.029,Y -514.603,Z 1334.655,A 0.000,B 0.000,C 90.000,E1 333.819} C_DIS
LIN {X -0.250,Y -512.638,Z 1334.651,A 0.000,B 0.000,C 90.000,E1 333.256} C_DIS
LIN {X 0.201,Y -510.361,Z 1334.648,A 0.000,B 0.000,C 90.000,E1 332.615} C_DIS
LIN {X -0.330,Y -508.300,Z 1334.646,A 0.000,B 0.000,C 90.000,E1 332.231} C_DIS
LIN {X -0.003,Y -506.645,Z 1334.644,A 0.000,B 0.000,C 90.000,E1 331.897} C_DIS
LIN {X -0.184,Y -505.674,Z 1334.643,A 0.000,B 0.000,C 90.000,E1 331.769} C_DIS
LIN {X 0.077,Y -504.506,Z 1334.642,A 0.000,B 0.000,C 90.000,E1 331.591} C_DIS
LIN {X 0.134,Y -502.863,Z 1334.641,A 0.000,B 0.000,C 90.000,E1 331.435} C_DIS
LIN {X -0.088,Y -476.383,Z 1334.632,A 0.000,B 0.000,C 90.000,E1 329.744} C_DIS
LIN {X 0.186,Y -452.940,Z 1334.622,A 0.000,B 0.000,C 90.000,E1 327.995} C_DIS
LIN {X -0.291,Y -431.483,Z 1334.613,A 0.000,B 0.000,C 90.000,E1 326.294} C_DIS
LIN {X -0.056,Y -410.494,Z 1334.602,A 0.000,B 0.000,C 90.000,E1 324.322} C_DIS
LIN {X -0.121,Y -391.491,Z 1334.591,A 0.000,B 0.000,C 90.000,E1 322.351} C_DIS
LIN {X 0.091,Y -374.720,Z 1334.580,A 0.000,B 0.000,C 90.000,E1 320.356} C_DIS
LIN {X 0.056,Y -374.721,Z 1334.580,A 0.000,B 0.000,C 90.000,E1 320.356} C_DIS
LIN {X 0.135,Y -378.165,Z 1334.563,A 0.000,B 0.000,C 90.000,E1 317.391} C_DIS
LIN {X 0.121,Y -383.807,Z 1334.531,A 0.000,B 0.000,C 90.000,E1 311.595} C_DIS
LIN {X -0.085,Y -384.798,Z 1334.527,A 0.000,B 0.000,C 90.000,E1 310.906} C_DIS
LIN {X -0.095,Y -390.967,Z 1334.493,A 0.000,B 0.000,C 90.000,E1 304.818} C_DIS
LIN {X -0.028,Y -391.372,Z 1334.491,A 0.000,B 0.000,C 90.000,E1 304.452} C_DIS
LIN {X 0.049,Y -396.699,Z 1334.460,A 0.000,B 0.000,C 90.000,E1 298.771} C_DIS
LIN {X -0.080,Y -397.078,Z 1334.458,A 0.000,B 0.000,C 90.000,E1 298.437} C_DIS
LIN {X -0.124,Y -401.498,Z 1334.427,A 0.000,B 0.000,C 90.000,E1 292.823} C_DIS
LIN {X 0.042,Y -401.770,Z 1334.423,A 0.000,B 0.000,C 90.000,E1 292.099} C_DIS
LIN {X 0.002,Y -404.574,Z 1334.396,A 0.000,B 0.000,C 90.000,E1 287.221} C_DIS
LIN {X 0.103,Y -404.760,Z 1334.394,A 0.000,B 0.000,C 90.000,E1 286.858} C_DIS
LIN {X 0.010,Y -406.044,Z 1334.365,A 0.000,B 0.000,C 90.000,E1 281.658} C_DIS
LIN {X 0.100,Y -406.134,Z 1334.363,A 0.000,B 0.000,C 90.000,E1 281.299} C_DIS
LIN {X 0.129,Y -405.657,Z 1334.334,A 0.000,B 0.000,C 90.000,E1 276.087} C_DIS
LIN {X 0.135,Y -405.594,Z 1334.332,A 0.000,B 0.000,C 90.000,E1 275.739} C_DIS
LIN {X -0.195,Y -403.547,Z 1334.305,A 0.000,B 0.000,C 90.000,E1 270.917} C_DIS
LIN {X 0.143,Y -403.030,Z 1334.301,A 0.000,B 0.000,C 90.000,E1 270.172} C_DIS
LIN {X -0.034,Y -399.005,Z 1334.272,A 0.000,B 0.000,C 90.000,E1 264.951} C_DIS
LIN {X -0.041,Y -394.756,Z 1334.252,A 0.000,B 0.000,C 90.000,E1 261.432} C_DIS
LIN {X 0.126,Y -392.916,Z 1334.241,A 0.000,B 0.000,C 90.000,E1 259.285} C_DIS
LIN {X 0.117,Y -391.853,Z 1334.237,A 0.000,B 0.000,C 90.000,E1 258.578} C_DIS
LIN {X -0.128,Y -385.722,Z 1334.211,A 0.000,B 0.000,C 90.000,E1 253.976} C_DIS
LIN {X -0.192,Y -384.950,Z 1334.207,A 0.000,B 0.000,C 90.000,E1 253.268} C_DIS
LIN {X 0.036,Y -378.101,Z 1334.183,A 0.000,B 0.000,C 90.000,E1 248.901} C_DIS
LIN {X -0.228,Y -376.343,Z 1334.175,A 0.000,B 0.000,C 90.000,E1 247.486} C_DIS
LIN {X -0.104,Y -375.833,Z 1334.173,A 0.000,B 0.000,C 90.000,E1 247.102} C_DIS
LIN {X 0.015,Y -369.069,Z 1334.150,A 0.000,B 0.000,C 90.000,E1 243.050} C_DIS
LIN {X -0.073,Y -366.221,Z 1334.138,A 0.000,B 0.000,C 90.000,E1 240.845} C_DIS
LIN {X 0.087,Y -358.816,Z 1334.113,A 0.000,B 0.000,C 90.000,E1 236.342} C_DIS
LIN {X -0.122,Y -356.007,Z 1334.101,A 0.000,B 0.000,C 90.000,E1 234.116} C_DIS
LIN {X -0.027,Y -348.927,Z 1334.075,A 0.000,B 0.000,C 90.000,E1 229.542} C_DIS
LIN {X -0.063,Y -345.856,Z 1334.060,A 0.000,B 0.000,C 90.000,E1 226.863} C_DIS
LIN {X 0.169,Y -342.381,Z 1334.047,A 0.000,B 0.000,C 90.000,E1 224.514} C_DIS
LIN {X 0.151,Y -342.381,Z 1334.047,A 0.000,B 0.000,C 90.000,E1 224.514} C_DIS
LIN {X -0.054,Y -358.020,Z 1334.034,A 0.000,B 0.000,C 90.000,E1 222.204} C_DIS
LIN {X 0.049,Y -374.798,Z 1334.022,A 0.000,B 0.000,C 90.000,E1 219.967} C_DIS
LIN {X -0.052,Y -392.230,Z 1334.011,A 0.000,B 0.000,C 90.000,E1 217.935} C_DIS
LIN {X 0.147,Y -411.631,Z 1334.000,A 0.000,B 0.000,C 90.000,E1 215.884} C_DIS
LIN {X 0.106,Y -433.056,Z 1333.989,A 0.000,B 0.000,C 90.000,E1 213.913} C_DIS
LIN {X 0.005,Y -443.954,Z 1333.983,A 0.000,B 0.000,C 90.000,E1 213.007} C_DIS
LIN {X 0.007,Y -445.903,Z 1333.982,A 0.000,B 0.000,C 90.000,E1 212.752} C_DIS
LIN {X 0.065,Y -447.376,Z 1333.980,A 0.000,B 0.000,C 90.000,E1 212.418} C_DIS
LIN {X 0.134,Y -448.479,Z 1333.978,A 0.000,B 0.000,C 90.000,E1 212.084} C_DIS
LIN {X -0.175,Y -449.372,Z 1333.977,A 0.000,B 0.000,C 90.000,E1 211.799} C_DIS
LIN {X -0.019,Y -450.782,Z 1333.973,A 0.000,B 0.000,C 90.000,E1 211.131} C_DIS
LIN {X 0.149,Y -451.860,Z 1333.969,A 0.000,B 0.000,C 90.000,E1 210.463} C_DIS
LIN {X -0.291,Y -452.658,Z 1333.966,A 0.000,B 0.000,C 90.000,E1 209.873} C_DIS
LIN {X 0.020,Y -457.410,Z 1333.944,A 0.000,B 0.000,C 90.000,E1 205.976} C_DIS
LIN {X -0.061,Y -459.688,Z 1333.936,A 0.000,B 0.000,C 90.000,E1 204.387} C_DIS
LIN {X 0.211,Y -461.389,Z 1333.928,A 0.000,B 0.000,C 90.000,E1 203.078} C_DIS
LIN {X -0.092,Y -463.056,Z 1333.921,A 0.000,B 0.000,C 90.000,E1 201.844} C_DIS
LIN {X 0.065,Y -464.757,Z 1333.914,A 0.000,B 0.000,C 90.000,E1 200.556} C_DIS
LIN {X 0.183,Y -466.707,Z 1333.906,A 0.000,B 0.000,C 90.000,E1 198.960} C_DIS
LIN {X 0.033,Y -468.632,Z 1333.897,A 0.000,B 0.000,C 90.000,E1 197.402} C_DIS
LIN {X 0.111,Y -470.070,Z 1333.890,A 0.000,B 0.000,C 90.000,E1 196.134} C_DIS
LIN {X -0.048,Y -471.495,Z 1333.883,A 0.000,B 0.000,C 90.000,E1 194.898} C_DIS
LIN {X 0.053,Y -473.551,Z 1333.872,A 0.000,B 0.000,C 90.000,E1 193.008} C_DIS
LIN {X -0.067,Y -476.020,Z 1333.860,A 0.000,B 0.000,C 90.000,E1 190.838} C_DIS
LIN {X 0.084,Y -477.771,Z 1333.852,A 0.000,B 0.000,C 90.000,E1 189.265} C_DIS
LIN {X -0.132,Y -479.096,Z 1333.845,A 0.000,B 0.000,C 90.000,E1 188.049} C_DIS
LIN {X -0.006,Y -480.570,Z 1333.836,A 0.000,B 0.000,C 90.000,E1 186.486} C_DIS
LIN {X 0.041,Y -481.764,Z 1333.828,A 0.000,B 0.000,C 90.000,E1 184.935} C_DIS
LIN {X -0.175,Y -482.548,Z 1333.821,A 0.000,B 0.000,C 90.000,E1 183.726} C_DIS
LIN {X 0.068,Y -483.071,Z 1333.814,A 0.000,B 0.000,C 90.000,E1 182.465} C_DIS
LIN {X 0.137,Y -483.357,Z 1333.805,A 0.000,B 0.000,C 90.000,E1 180.917} C_DIS
LIN {X 0.079,Y -483.330,Z 1333.800,A 0.000,B 0.000,C 90.000,E1 180.000} C_DIS
LIN {X -0.162,Y -483.093,Z 1333.793,A 0.000,B 0.000,C 90.000,E1 178.797} C_DIS
LIN {X 0.087,Y -482.565,Z 1333.786,A 0.000,B 0.000,C 90.000,E1 177.535} C_DIS
LIN {X 0.035,Y -481.968,Z 1333.781,A 0.000,B 0.000,C 90.000,E1 176.617} C_DIS
LIN {X -0.216,Y -480.721,Z 1333.774,A 0.000,B 0.000,C 90.000,E1 175.412} C_DIS
LIN {X 0.026,Y -479.094,Z 1333.768,A 0.000,B 0.000,C 90.000,E1 174.147} C_DIS
LIN {X -0.022,Y -477.530,Z 1333.762,A 0.000,B 0.000,C 90.000,E1 173.223} C_DIS
LIN {X 0.075,Y -476.202,Z 1333.759,A 0.000,B 0.000,C 90.000,E1 172.591} C_DIS
LIN {X 0.061,Y -473.811,Z 1333.754,A 0.000,B 0.000,C 90.000,E1 171.659} C_DIS
LIN {X -0.174,Y -472.919,Z 1333.752,A 0.000,B 0.000,C 90.000,E1 171.376} C_DIS
LIN {X -0.046,Y -470.664,Z 1333.749,A 0.000,B 0.000,C 90.000,E1 170.735} C_DIS
LIN {X 0.163,Y -467.495,Z 1333.744,A 0.000,B 0.000,C 90.000,E1 169.926} C_DIS
LIN {X 0.045,Y -462.420,Z 1333.739,A 0.000,B 0.000,C 90.000,E1 168.993} C_DIS
LIN {X -0.035,Y -456.569,Z 1333.734,A 0.000,B 0.000,C 90.000,E1 168.049} C_DIS
LIN {X 0.068,Y -447.291,Z 1333.726,A 0.000,B 0.000,C 90.000,E1 166.589} C_DIS
LIN {X -0.199,Y -436.834,Z 1333.717,A 0.000,B 0.000,C 90.000,E1 164.991} C_DIS
LIN {X 0.073,Y -428.459,Z 1333.709,A 0.000,B 0.000,C 90.000,E1 163.630} C_DIS
LIN {X 0.073,Y -424.934,Z 1333.705,A 0.000,B 0.000,C 90.000,E1 162.960} C_DIS
LIN {X 0.171,Y -424.171,Z 1333.704,A 0.000,B 0.000,C 90.000,E1 162.779} C_DIS
LIN {X 0.125,Y -422.709,Z 1333.701,A 0.000,B 0.000,C 90.000,E1 162.181} C_DIS
LIN {X -0.208,Y -422.515,Z 1333.700,A 0.000,B 0.000,C 90.000,E1 161.945} C_DIS
LIN {X 0.064,Y -422.767,Z 1333.699,A 0.000,B 0.000,C 90.000,E1 161.764} C_DIS
LIN {X -0.016,Y -424.268,Z 1333.697,A 0.000,B 0.000,C 90.000,E1 161.511} C_DIS
LIN {X 0.206,Y -425.140,Z 1333.696,A 0.000,B 0.000,C 90.000,E1 161.275} C_DIS
LIN {X 0.167,Y -425.183,Z 1333.696,A 0.000,B 0.000,C 90.000,E1 161.275} C_DIS
LIN {X 0.172,Y -426.545,Z 1333.695,A 0.000,B 0.000,C 90.000,E1 161.148} C_DIS
LIN {X -0.091,Y -429.609,Z 1333.694,A 0.000,B 0.000,C 90.000,E1 160.859} C_DIS
LIN {X -0.069,Y -434.576,Z 1333.691,A 0.000,B 0.000,C 90.000,E1 160.423} C_DIS
LIN {X 0.142,Y -440.407,Z 1333.689,A 0.000,B 0.000,C 90.000,E1 159.934} C_DIS
LIN {X 0.072,Y -454.556,Z 1333.683,A 0.000,B 0.000,C 90.000,E1 158.847} C_DIS
LIN {X -0.203,Y -468.601,Z 1333.677,A 0.000,B 0.000,C 90.000,E1 157.794} C_DIS
LIN {X -0.155,Y -477.727,Z 1333.672,A 0.000,B 0.000,C 90.000,E1 157.050} C_DIS
LIN {X -0.094,Y -483.600,Z 1333.670,A 0.000,B 0.000,C 90.000,E1 156.538} C_DIS
LIN {X -0.205,Y -487.804,Z 1333.668,A 0.000,B 0.000,C 90.000,E1 156.177} C_DIS
LIN {X 0.025,Y -494.856,Z 1333.664,A 0.000,B 0.000,C 90.000,E1 155.485} C_DIS
LIN {X -0.036,Y -498.856,Z 1333.662,A 0.000,B 0.000,C 90.000,E1 155.101} C_DIS
LIN {X -0.195,Y -506.978,Z 1333.657,A 0.000,B 0.000,C 90.000,E1 154.280} C_DIS
LIN {X -0.062,Y -513.214,Z 1333.653,A 0.000,B 0.000,C 90.000,E1 153.563} C_DIS
LIN {X -0.123,Y -516.987,Z 1333.651,A 0.000,B 0.000,C 90.000,E1 153.127} C_DIS
LIN {X -0.096,Y -521.601,Z 1333.647,A 0.000,B 0.000,C 90.000,E1 152.538} C_DIS
LIN {X -0.036,Y -525.711,Z 1333.644,A 0.000,B 0.000,C 90.000,E1 151.948} C_DIS
LIN {X -0.195,Y -529.312,Z 1333.641,A 0.000,B 0.000,C 90.000,E1 151.385} C_DIS
LIN {X -0.228,Y -532.935,Z 1333.637,A 0.000,B 0.000,C 90.000,E1 150.667} C_DIS
LIN {X -0.087,Y -535.294,Z 1333.634,A 0.000,B 0.000,C 90.000,E1 150.078} C_DIS
LIN {X 0.070,Y -537.306,Z 1333.631,A 0.000,B 0.000,C 90.000,E1 149.488} C_DIS
LIN {X -0.223,Y -539.860,Z 1333.626,A 0.000,B 0.000,C 90.000,E1 148.663} C_DIS
LIN {X -0.023,Y -542.070,Z 1333.621,A 0.000,B 0.000,C 90.000,E1 147.788} C_DIS
LIN {X 0.201,Y -543.923,Z 1333.616,A 0.000,B 0.000,C 90.000,E1 146.914} C_DIS
LIN {X 0.021,Y -545.954,Z 1333.610,A 0.000,B 0.000,C 90.000,E1 145.801} C_DIS
LIN {X -0.172,Y -547.106,Z 1333.605,A 0.000,B 0.000,C 90.000,E1 144.975} C_DIS
LIN {X -0.038,Y -548.040,Z 1333.601,A 0.000,B 0.000,C 90.000,E1 144.116} C_DIS
LIN {X 0.163,Y -548.985,Z 1333.594,A 0.000,B 0.000,C 90.000,E1 142.970} C_DIS
LIN {X 0.110,Y -550.229,Z 1333.583,A 0.000,B 0.000,C 90.000,E1 141.009} C_DIS
LIN {X 0.061,Y -551.871,Z 1333.571,A 0.000,B 0.000,C 90.000,E1 138.771} C_DIS
LIN {X -0.244,Y -552.578,Z 1333.568,A 0.000,B 0.000,C 90.000,E1 138.243} C_DIS
LIN {X 0.149,Y -553.552,Z 1333.565,A 0.000,B 0.000,C 90.000,E1 137.634} C_DIS
LIN {X 0.106,Y -553.578,Z 1333.565,A 0.000,B 0.000,C 90.000,E1 137.634} C_DIS
LIN {X 0.038,Y -554.339,Z 1333.564,A 0.000,B 0.000,C 90.000,E1 137.514} C_DIS
LIN {X -0.122,Y -557.228,Z 1333.563,A 0.000,B 0.000,C 90.000,E1 137.391} C_DIS
LIN {X -0.114,Y -559.598,Z 1333.563,A 0.000,B 0.000,C 90.000,E1 137.310} C_DIS
LIN {X -0.027,Y -569.329,Z 1333.561,A 0.000,B 0.000,C 90.000,E1 137.025} C_DIS
LIN {X 0.116,Y -572.763,Z 1333.561,A 0.000,B 0.000,C 90.000,E1 136.905} C_DIS
LIN {X -0.161,Y -575.328,Z 1333.560,A 0.000,B 0.000,C 90.000,E1 136.824} C_DIS
LIN {X 0.022,Y -578.355,Z 1333.559,A 0.000,B 0.000,C 90.000,E1 136.662} C_DIS
LIN {X 0.301,Y -584.273,Z 1333.557,A 0.000,B 0.000,C 90.000,E1 136.296} C_DIS
LIN {X -0.388,Y -589.959,Z 1333.555,A 0.000,B 0.000,C 90.000,E1 135.972} C_DIS
LIN {X 0.158,Y -595.392,Z 1333.553,A 0.000,B 0.000,C 90.000,E1 135.486} C_DIS
LIN {X -0.076,Y -600.685,Z 1333.550,A 0.000,B 0.000,C 90.000,E1 135.040} C_DIS
LIN {X -0.073,Y -604.645,Z 1333.548,A 0.000,B 0.000,C 90.000,E1 134.676} C_DIS
LIN {X 0.277,Y -608.390,Z 1333.546,A 0.000,B 0.000,C 90.000,E1 134.271} C_DIS
LIN {X 0.190,Y -616.353,Z 1333.541,A 0.000,B 0.000,C 90.000,E1 133.380} C_DIS
LIN {X 0.021,Y -624.702,Z 1333.535,A 0.000,B 0.000,C 90.000,E1 132.366} C_DIS
LIN {X -0.298,Y -629.404,Z 1333.532,A 0.000,B 0.000,C 90.000,E1 131.757} C_DIS
LIN {X -0.073,Y -633.102,Z 1333.529,A 0.000,B 0.000,C 90.000,E1 131.229} C_DIS
LIN {X 0.074,Y -638.568,Z 1333.525,A 0.000,B 0.000,C 90.000,E1 130.458} C_DIS
LIN {X -0.131,Y -645.405,Z 1333.519,A 0.000,B 0.000,C 90.000,E1 129.483} C_DIS
LIN {X -0.336,Y -652.545,Z 1333.513,A 0.000,B 0.000,C 90.000,E1 128.382} C_DIS
LIN {X 0.048,Y -658.599,Z 1333.508,A 0.000,B 0.000,C 90.000,E1 127.363} C_DIS
LIN {X 0.117,Y -664.086,Z 1333.502,A 0.000,B 0.000,C 90.000,E1 126.377} C_DIS
LIN {X -0.303,Y -667.194,Z 1333.499,A 0.000,B 0.000,C 90.000,E1 125.804} C_DIS
LIN {X 0.290,Y -670.568,Z 1333.495,A 0.000,B 0.000,C 90.000,E1 125.025} C_DIS
LIN {X -0.020,Y -673.610,Z 1333.491,A 0.000,B 0.000,C 90.000,E1 124.326} C_DIS
LIN {X 0.099,Y -675.458,Z 1333.488,A 0.000,B 0.000,C 90.000,E1 123.833} C_DIS
LIN {X 0.396,Y -677.827,Z 1333.484,A 0.000,B 0.000,C 90.000,E1 123.086} C_DIS
LIN {X 0.327,Y -680.525,Z 1333.479,A 0.000,B 0.000,C 90.000,E1 122.133} C_DIS
LIN {X -0.262,Y -682.292,Z 1333.475,A 0.000,B 0.000,C 90.000,E1 121.465} C_DIS
LIN {X 0.102,Y -683.829,Z 1333.471,A 0.000,B 0.000,C 90.000,E1 120.718} C_DIS
LIN {X 0.133,Y -685.144,Z 1333.467,A 0.000,B 0.000,C 90.000,E1 120.001} C_DIS
LIN {X 0.182,Y -686.123,Z 1333.463,A 0.000,B 0.000,C 90.000,E1 119.283} C_DIS
LIN {X 0.021,Y -686.638,Z 1333.460,A 0.000,B 0.000,C 90.000,E1 118.821} C_DIS
LIN {X 0.085,Y -687.105,Z 1333.456,A 0.000,B 0.000,C 90.000,E1 118.103} C_DIS
LIN {X 0.378,Y -687.324,Z 1333.451,A 0.000,B 0.000,C 90.000,E1 117.129} C_DIS
LIN {X 0.136,Y -687.316,Z 1333.447,A 0.000,B 0.000,C 90.000,E1 116.437} C_DIS
LIN {X 0.199,Y -687.009,Z 1333.443,A 0.000,B 0.000,C 90.000,E1 115.720} C_DIS
LIN {X -0.266,Y -686.657,Z 1333.440,A 0.000,B 0.000,C 90.000,E1 115.283} C_DIS
LIN {X 0.181,Y -686.011,Z 1333.438,A 0.000,B 0.000,C 90.000,E1 114.771} C_DIS
LIN {X -0.286,Y -685.035,Z 1333.435,A 0.000,B 0.000,C 90.000,E1 114.335} C_DIS
LIN {X -0.069,Y -684.440,Z 1333.434,A 0.000,B 0.000,C 90.000,E1 114.079} C_DIS
LIN {X 0.188,Y -681.738,Z 1333.431,A 0.000,B 0.000,C 90.000,E1 113.462} C_DIS
LIN {X 0.291,Y -680.857,Z 1333.430,A 0.000,B 0.000,C 90.000,E1 113.334} C_DIS
LIN {X -0.204,Y -676.304,Z 1333.427,A 0.000,B 0.000,C 90.000,E1 112.898} C_DIS
LIN {X -0.111,Y -674.643,Z 1333.427,A 0.000,B 0.000,C 90.000,E1 112.770} C_DIS
LIN {X 0.183,Y -667.332,Z 1333.425,A 0.000,B 0.000,C 90.000,E1 112.386} C_DIS
LIN {X -0.121,Y -665.120,Z 1333.424,A 0.000,B 0.000,C 90.000,E1 112.333} C_DIS
LIN {X 0.015,Y -658.820,Z 1333.423,A 0.000,B 0.000,C 90.000,E1 112.153} C_DIS
LIN {X -0.110,Y -650.191,Z 1333.422,A 0.000,B 0.000,C 90.000,E1 112.025} C_DIS
LIN {X -0.144,Y -644.497,Z 1333.422,A 0.000,B 0.000,C 90.000,E1 111.950} C_DIS
LIN {X 0.196,Y -641.254,Z 1333.422,A 0.000,B 0.000,C 90.000,E1 111.844} C_DIS
LIN {X 0.160,Y -641.165,Z 1333.422,A 0.000,B 0.000,C 90.000,E1 111.844} C_DIS
LIN {X 0.034,Y -642.861,Z 1333.420,A 0.000,B 0.000,C 90.000,E1 111.589} C_DIS
LIN {X 0.183,Y -648.201,Z 1333.416,A 0.000,B 0.000,C 90.000,E1 110.918} C_DIS
LIN {X 0.065,Y -651.106,Z 1333.414,A 0.000,B 0.000,C 90.000,E1 110.556} C_DIS
LIN {X 0.096,Y -656.022,Z 1333.410,A 0.000,B 0.000,C 90.000,E1 109.812} C_DIS
LIN {X -0.102,Y -659.532,Z 1333.407,A 0.000,B 0.000,C 90.000,E1 109.214} C_DIS
LIN {X -0.111,Y -661.933,Z 1333.404,A 0.000,B 0.000,C 90.000,E1 108.725} C_DIS
LIN {X -0.205,Y -665.162,Z 1333.400,A 0.000,B 0.000,C 90.000,E1 108.000} C_DIS
LIN {X -0.272,Y -667.964,Z 1333.396,A 0.000,B 0.000,C 90.000,E1 107.275} C_DIS
LIN {X 0.327,Y -670.498,Z 1333.392,A 0.000,B 0.000,C 90.000,E1 106.496} C_DIS
LIN {X 0.122,Y -672.610,Z 1333.388,A 0.000,B 0.000,C 90.000,E1 105.788} C_DIS
LIN {X 0.119,Y -674.449,Z 1333.384,A 0.000,B 0.000,C 90.000,E1 105.064} C_DIS
LIN {X -0.047,Y -676.003,Z 1333.380,A 0.000,B 0.000,C 90.000,E1 104.356} C_DIS
LIN {X -0.197,Y -677.092,Z 1333.376,A 0.000,B 0.000,C 90.000,E1 103.647} C_DIS
LIN {X -0.292,Y -677.649,Z 1333.373,A 0.000,B 0.000,C 90.000,E1 103.175} C_DIS
LIN {X 0.042,Y -678.016,Z 1333.368,A 0.000,B 0.000,C 90.000,E1 102.187} C_DIS
LIN {X -0.046,Y -677.994,Z 1333.365,A 0.000,B 0.000,C 90.000,E1 101.715} C_DIS
LIN {X -0.091,Y -677.942,Z 1333.364,A 0.000,B 0.000,C 90.000,E1 101.478} C_DIS
LIN {X -0.361,Y -677.254,Z 1333.360,A 0.000,B 0.000,C 90.000,E1 100.782} C_DIS
LIN {X 0.206,Y -676.590,Z 1333.357,A 0.000,B 0.000,C 90.000,E1 100.254} C_DIS
LIN {X -0.018,Y -675.722,Z 1333.354,A 0.000,B 0.000,C 90.000,E1 99.792} C_DIS
LIN {X -0.134,Y -674.570,Z 1333.352,A 0.000,B 0.000,C 90.000,E1 99.321} C_DIS
LIN {X 0.299,Y -673.042,Z 1333.349,A 0.000,B 0.000,C 90.000,E1 98.803} C_DIS
LIN {X 0.061,Y -671.231,Z 1333.346,A 0.000,B 0.000,C 90.000,E1 98.341} C_DIS
LIN {X -0.269,Y -668.129,Z 1333.342,A 0.000,B 0.000,C 90.000,E1 97.644} C_DIS
LIN {X 0.029,Y -664.557,Z 1333.338,A 0.000,B 0.000,C 90.000,E1 96.891} C_DIS
LIN {X 0.205,Y -660.725,Z 1333.334,A 0.000,B 0.000,C 90.000,E1 96.144} C_DIS
LIN {X -0.209,Y -657.123,Z 1333.331,A 0.000,B 0.000,C 90.000,E1 95.568} C_DIS
LIN {X -0.100,Y -652.215,Z 1333.327,A 0.000,B 0.000,C 90.000,E1 94.821} C_DIS
LIN {X 0.179,Y -648.695,Z 1333.324,A 0.000,B 0.000,C 90.000,E1 94.302} C_DIS
LIN {X -0.216,Y -644.988,Z 1333.321,A 0.000,B 0.000,C 90.000,E1 93.841} C_DIS
LIN {X -0.032,Y -640.976,Z 1333.318,A 0.000,B 0.000,C 90.000,E1 93.326} C_DIS
LIN {X 0.159,Y -636.516,Z 1333.316,A 0.000,B 0.000,C 90.000,E1 92.808} C_DIS
LIN {X 0.239,Y -630.368,Z 1333.312,A 0.000,B 0.000,C 90.000,E1 92.178} C_DIS
LIN {X 0.195,Y -620.285,Z 1333.307,A 0.000,B 0.000,C 90.000,E1 91.203} C_DIS
LIN {X 0.094,Y -616.424,Z 1333.305,A 0.000,B 0.000,C 90.000,E1 90.859} C_DIS
LIN {X 0.201,Y -609.547,Z 1333.302,A 0.000,B 0.000,C 90.000,E1 90.286} C_DIS
LIN {X 0.071,Y -602.903,Z 1333.299,A 0.000,B 0.000,C 90.000,E1 89.885} C_DIS
LIN {X -0.026,Y -596.037,Z 1333.297,A 0.000,B 0.000,C 90.000,E1 89.542} C_DIS
LIN {X -0.236,Y -588.997,Z 1333.296,A 0.000,B 0.000,C 90.000,E1 89.255} C_DIS
LIN {X 0.273,Y -578.967,Z 1333.293,A 0.000,B 0.000,C 90.000,E1 88.797} C_DIS
LIN {X 0.119,Y -577.399,Z 1333.293,A 0.000,B 0.000,C 90.000,E1 88.740} C_DIS
LIN {X -0.039,Y -573.400,Z 1333.291,A 0.000,B 0.000,C 90.000,E1 88.453} C_DIS
LIN {X 0.149,Y -573.079,Z 1333.291,A 0.000,B 0.000,C 90.000,E1 88.396} C_DIS
LIN {X 0.115,Y -573.069,Z 1333.291,A 0.000,B 0.000,C 90.000,E1 88.396} C_DIS
LIN {X -0.228,Y -572.497,Z 1333.290,A 0.000,B 0.000,C 90.000,E1 88.224} C_DIS
LIN {X 0.146,Y -572.279,Z 1333.289,A 0.000,B 0.000,C 90.000,E1 88.051} C_DIS
LIN {X -0.009,Y -572.234,Z 1333.287,A 0.000,B 0.000,C 90.000,E1 87.650} C_DIS
LIN {X -0.114,Y -575.019,Z 1333.270,A 0.000,B 0.000,C 90.000,E1 84.666} C_DIS
LIN {X 0.138,Y -577.562,Z 1333.258,A 0.000,B 0.000,C 90.000,E1 82.470} C_DIS
LIN {X 0.116,Y -579.513,Z 1333.249,A 0.000,B 0.000,C 90.000,E1 80.849} C_DIS
LIN {X -0.002,Y -581.109,Z 1333.242,A 0.000,B 0.000,C 90.000,E1 79.511} C_DIS
LIN {X -0.100,Y -582.544,Z 1333.234,A 0.000,B 0.000,C 90.000,E1 78.173} C_DIS
LIN {X -0.065,Y -583.753,Z 1333.227,A 0.000,B 0.000,C 90.000,E1 76.825} C_DIS
LIN {X 0.129,Y -584.822,Z 1333.219,A 0.000,B 0.000,C 90.000,E1 75.463} C_DIS
LIN {X -0.147,Y -586.110,Z 1333.209,A 0.000,B 0.000,C 90.000,E1 73.614} C_DIS
LIN {X 0.171,Y -586.658,Z 1333.204,A 0.000,B 0.000,C 90.000,E1 72.779} C_DIS
LIN {X -0.218,Y -588.045,Z 1333.193,A 0.000,B 0.000,C 90.000,E1 70.678} C_DIS
LIN {X -0.193,Y -589.376,Z 1333.181,A 0.000,B 0.000,C 90.000,E1 68.539} C_DIS
LIN {X 0.098,Y -590.206,Z 1333.173,A 0.000,B 0.000,C 90.000,E1 67.177} C_DIS
LIN {X -0.246,Y -591.340,Z 1333.164,A 0.000,B 0.000,C 90.000,E1 65.613} C_DIS
LIN {X -0.119,Y -592.094,Z 1333.159,A 0.000,B 0.000,C 90.000,E1 64.537} C_DIS
LIN {X -0.082,Y -593.078,Z 1333.151,A 0.000,B 0.000,C 90.000,E1 63.204} C_DIS
LIN {X 0.146,Y -595.009,Z 1333.138,A 0.000,B 0.000,C 90.000,E1 60.795} C_DIS
LIN {X 0.308,Y -597.071,Z 1333.126,A 0.000,B 0.000,C 90.000,E1 58.663} C_DIS
LIN {X 0.107,Y -598.986,Z 1333.116,A 0.000,B 0.000,C 90.000,E1 56.834} C_DIS
LIN {X 0.132,Y -600.338,Z 1333.109,A 0.000,B 0.000,C 90.000,E1 55.515} C_DIS
LIN {X -0.070,Y -601.393,Z 1333.103,A 0.000,B 0.000,C 90.000,E1 54.482} C_DIS
LIN {X 0.004,Y -603.146,Z 1333.093,A 0.000,B 0.000,C 90.000,E1 52.637} C_DIS
LIN {X -0.040,Y -604.080,Z 1333.085,A 0.000,B 0.000,C 90.000,E1 51.331} C_DIS
LIN {X 0.054,Y -604.819,Z 1333.079,A 0.000,B 0.000,C 90.000,E1 50.275} C_DIS
LIN {X 0.164,Y -605.415,Z 1333.074,A 0.000,B 0.000,C 90.000,E1 49.218} C_DIS
LIN {X 0.281,Y -605.783,Z 1333.068,A 0.000,B 0.000,C 90.000,E1 48.162} C_DIS
LIN {X 0.143,Y -605.931,Z 1333.063,A 0.000,B 0.000,C 90.000,E1 47.391} C_DIS
LIN {X 0.284,Y -606.156,Z 1333.055,A 0.000,B 0.000,C 90.000,E1 45.810} C_DIS
LIN {X -0.052,Y -606.139,Z 1333.049,A 0.000,B 0.000,C 90.000,E1 44.798} C_DIS
LIN {X -0.196,Y -605.998,Z 1333.045,A 0.000,B 0.000,C 90.000,E1 44.028} C_DIS
LIN {X 0.082,Y -605.752,Z 1333.040,A 0.000,B 0.000,C 90.000,E1 43.218} C_DIS
LIN {X -0.200,Y -605.178,Z 1333.031,A 0.000,B 0.000,C 90.000,E1 41.676} C_DIS
LIN {X 0.168,Y -604.620,Z 1333.024,A 0.000,B 0.000,C 90.000,E1 40.334} C_DIS
LIN {X 0.319,Y -603.831,Z 1333.016,A 0.000,B 0.000,C 90.000,E1 38.749} C_DIS
LIN {X -0.230,Y -603.379,Z 1333.011,A 0.000,B 0.000,C 90.000,E1 38.016} C_DIS
LIN {X -0.049,Y -602.561,Z 1333.005,A 0.000,B 0.000,C 90.000,E1 36.950} C_DIS
LIN {X 0.123,Y -601.185,Z 1333.000,A 0.000,B 0.000,C 90.000,E1 35.884} C_DIS
LIN {X 0.030,Y -599.946,Z 1332.995,A 0.000,B 0.000,C 90.000,E1 35.105} C_DIS
LIN {X 0.157,Y -598.119,Z 1332.989,A 0.000,B 0.000,C 90.000,E1 34.040} C_DIS
LIN {X 0.289,Y -597.074,Z 1332.986,A 0.000,B 0.000,C 90.000,E1 33.499} C_DIS
LIN {X -0.066,Y -594.034,Z 1332.979,A 0.000,B 0.000,C 90.000,E1 32.212} C_DIS
LIN {X 0.042,Y -592.621,Z 1332.976,A 0.000,B 0.000,C 90.000,E1 31.671} C_DIS
LIN {X 0.227,Y -589.291,Z 1332.970,A 0.000,B 0.000,C 90.000,E1 30.590} C_DIS
LIN {X 0.181,Y -586.403,Z 1332.966,A 0.000,B 0.000,C 90.000,E1 29.795} C_DIS
LIN {X -0.057,Y -584.297,Z 1332.963,A 0.000,B 0.000,C 90.000,E1 29.283} C_DIS
LIN {X -0.153,Y -580.725,Z 1332.958,A 0.000,B 0.000,C 90.000,E1 28.487} C_DIS
LIN {X 0.091,Y -578.179,Z 1332.955,A 0.000,B 0.000,C 90.000,E1 27.924} C_DIS
LIN {X -0.079,Y -573.981,Z 1332.951,A 0.000,B 0.000,C 90.000,E1 27.129} C_DIS
LIN {X -0.046,Y -569.307,Z 1332.946,A 0.000,B 0.000,C 90.000,E1 26.309} C_DIS
LIN {X 0.278,Y -565.069,Z 1332.942,A 0.000,B 0.000,C 90.000,E1 25.591} C_DIS
LIN {X 0.001,Y -562.374,Z 1332.940,A 0.000,B 0.000,C 90.000,E1 25.207} C_DIS
LIN {X 0.014,Y -557.498,Z 1332.936,A 0.000,B 0.000,C 90.000,E1 24.515} C_DIS
LIN {X 0.096,Y -553.442,Z 1332.933,A 0.000,B 0.000,C 90.000,E1 23.951} C_DIS
LIN {X 0.147,Y -549.038,Z 1332.930,A 0.000,B 0.000,C 90.000,E1 23.387} C_DIS
LIN {X -0.026,Y -543.443,Z 1332.926,A 0.000,B 0.000,C 90.000,E1 22.717} C_DIS
LIN {X 0.184,Y -533.815,Z 1332.920,A 0.000,B 0.000,C 90.000,E1 21.589} C_DIS
LIN {X -0.006,Y -523.281,Z 1332.914,A 0.000,B 0.000,C 90.000,E1 20.482} C_DIS
LIN {X -0.185,Y -512.733,Z 1332.908,A 0.000,B 0.000,C 90.000,E1 19.396} C_DIS
LIN {X -0.211,Y -503.411,Z 1332.902,A 0.000,B 0.000,C 90.000,E1 18.417} C_DIS
LIN {X -0.062,Y -492.502,Z 1332.896,A 0.000,B 0.000,C 90.000,E1 17.330} C_DIS
LIN {X -0.005,Y -478.187,Z 1332.889,A 0.000,B 0.000,C 90.000,E1 15.969} C_DIS
LIN {X -0.189,Y -466.611,Z 1332.883,A 0.000,B 0.000,C 90.000,E1 14.898} C_DIS
LIN {X 0.065,Y -452.043,Z 1332.875,A 0.000,B 0.000,C 90.000,E1 13.480} C_DIS
LIN {X 0.114,Y -427.849,Z 1332.861,A 0.000,B 0.000,C 90.000,E1 11.007} C_DIS
LIN {X 0.072,Y -415.027,Z 1332.854,A 0.000,B 0.000,C 90.000,E1 9.613} C_DIS
LIN {X 0.015,Y -403.671,Z 1332.846,A 0.000,B 0.000,C 90.000,E1 8.341} C_DIS
LIN {X -0.089,Y -399.487,Z 1332.844,A 0.000,B 0.000,C 90.000,E1 7.871} C_DIS
LIN {X 0.162,Y -395.470,Z 1332.841,A 0.000,B 0.000,C 90.000,E1 7.296} C_DIS
LIN {X 0.098,Y -395.199,Z 1332.840,A 0.000,B 0.000,C 90.000,E1 7.239} C_DIS
LIN {X 0.064,Y -395.202,Z 1332.840,A 0.000,B 0.000,C 90.000,E1 7.239} C_DIS
LIN {X -0.148,Y -395.439,Z 1332.840,A 0.000,B 0.000,C 90.000,E1 7.182} C_DIS
LIN {X -0.186,Y -395.480,Z 1332.840,A 0.000,B 0.000,C 90.000,E1 7.182} C_DIS
LIN {X 0.129,Y -399.924,Z 1332.838,A 0.000,B 0.000,C 90.000,E1 6.720} C_DIS
LIN {X 0.167,Y -412.155,Z 1332.833,A 0.000,B 0.000,C 90.000,E1 5.910} C_DIS
LIN {X -0.189,Y -417.138,Z 1332.831,A 0.000,B 0.000,C 90.000,E1 5.625} C_DIS
LIN {X 0.100,Y -423.428,Z 1332.828,A 0.000,B 0.000,C 90.000,E1 5.106} C_DIS
LIN {X 0.105,Y -429.551,Z 1332.826,A 0.000,B 0.000,C 90.000,E1 4.588} C_DIS
LIN {X 0.106,Y -436.963,Z 1332.822,A 0.000,B 0.000,C 90.000,E1 3.898} C_DIS
LIN {X -0.132,Y -444.161,Z 1332.818,A 0.000,B 0.000,C 90.000,E1 3.212} C_DIS
LIN {X 0.206,Y -449.806,Z 1332.815,A 0.000,B 0.000,C 90.000,E1 2.579} C_DIS
LIN {X -0.065,Y -455.265,Z 1332.811,A 0.000,B 0.000,C 90.000,E1 2.007} C_DIS
LIN {X -0.006,Y -461.534,Z 1332.807,A 0.000,B 0.000,C 90.000,E1 1.260} C_DIS
LIN {X -0.055,Y -466.558,Z 1332.803,A 0.000,B 0.000,C 90.000,E1 0.630} C_DIS
LIN {X -0.149,Y -470.149,Z 1332.801,A 0.000,B 0.000,C 90.000,E1 0.172} C_DIS
LIN {X 0.087,Y -475.920,Z 1332.796,A 0.000,B 0.000,C 90.000,E1 359.312} C_DIS
LIN {X -0.189,Y -480.899,Z 1332.792,A 0.000,B 0.000,C 90.000,E1 358.568} C_DIS
LIN {X 0.077,Y -485.456,Z 1332.788,A 0.000,B 0.000,C 90.000,E1 357.764} C_DIS
LIN {X -0.119,Y -489.779,Z 1332.783,A 0.000,B 0.000,C 90.000,E1 357.020} C_DIS
LIN {X 0.074,Y -493.020,Z 1332.780,A 0.000,B 0.000,C 90.000,E1 356.388} C_DIS
LIN {X -0.026,Y -496.677,Z 1332.776,A 0.000,B 0.000,C 90.000,E1 355.641} C_DIS
LIN {X 0.089,Y -500.741,Z 1332.771,A 0.000,B 0.000,C 90.000,E1 354.723} C_DIS
LIN {X 0.109,Y -503.927,Z 1332.767,A 0.000,B 0.000,C 90.000,E1 353.970} C_DIS
LIN {X -0.084,Y -506.251,Z 1332.763,A 0.000,B 0.000,C 90.000,E1 353.394} C_DIS
LIN {X 0.070,Y -510.554,Z 1332.757,A 0.000,B 0.000,C 90.000,E1 352.186} C_DIS
LIN {X -0.013,Y -512.534,Z 1332.753,A 0.000,B 0.000,C 90.000,E1 351.602} C_DIS
LIN {X -0.185,Y -515.109,Z 1332.748,A 0.000,B 0.000,C 90.000,E1 350.735} C_DIS
LIN {X 0.252,Y -518.220,Z 1332.742,A 0.000,B 0.000,C 90.000,E1 349.511} C_DIS
LIN {X 0.231,Y -520.851,Z 1332.735,A 0.000,B 0.000,C 90.000,E1 348.342} C_DIS
LIN {X 0.239,Y -522.602,Z 1332.731,A 0.000,B 0.000,C 90.000,E1 347.465} C_DIS
LIN {X -0.238,Y -524.594,Z 1332.724,A 0.000,B 0.000,C 90.000,E1 346.353} C_DIS
LIN {X -0.074,Y -525.812,Z 1332.719,A 0.000,B 0.000,C 90.000,E1 345.463} C_DIS
LIN {X 0.121,Y -527.092,Z 1332.713,A 0.000,B 0.000,C 90.000,E1 344.283} C_DIS
LIN {X -0.046,Y -527.733,Z 1332.708,A 0.000,B 0.000,C 90.000,E1 343.433} C_DIS
LIN {X -0.017,Y -528.075,Z 1332.705,A 0.000,B 0.000,C 90.000,E1 342.851} C_DIS
LIN {X 0.009,Y -528.297,Z 1332.698,A 0.000,B 0.000,C 90.000,E1 341.692} C_DIS
LIN {X -0.124,Y -528.095,Z 1332.692,A 0.000,B 0.000,C 90.000,E1 340.550} C_DIS
LIN {X -0.089,Y -527.284,Z 1332.686,A 0.000,B 0.000,C 90.000,E1 339.390} C_DIS
LIN {X 0.265,Y -526.587,Z 1332.682,A 0.000,B 0.000,C 90.000,E1 338.773} C_DIS
LIN {X -0.069,Y -525.789,Z 1332.679,A 0.000,B 0.000,C 90.000,E1 338.230} C_DIS
LIN {X -0.046,Y -524.284,Z 1332.674,A 0.000,B 0.000,C 90.000,E1 337.358} C_DIS
LIN {X -0.198,Y -523.257,Z 1332.671,A 0.000,B 0.000,C 90.000,E1 336.794} C_DIS
LIN {X -0.200,Y -521.401,Z 1332.666,A 0.000,B 0.000,C 90.000,E1 335.921} C_DIS
LIN {X -0.005,Y -519.194,Z 1332.661,A 0.000,B 0.000,C 90.000,E1 335.025} C_DIS
LIN {X 0.074,Y -515.730,Z 1332.655,A 0.000,B 0.000,C 90.000,E1 333.845} C_DIS
LIN {X 0.091,Y -512.020,Z 1332.648,A 0.000,B 0.000,C 90.000,E1 332.666} C_DIS
LIN {X -0.154,Y -509.949,Z 1332.645,A 0.000,B 0.000,C 90.000,E1 332.103} C_DIS
LIN {X -0.177,Y -507.502,Z 1332.642,A 0.000,B 0.000,C 90.000,E1 331.513} C_DIS
LIN {X -0.035,Y -505.247,Z 1332.639,A 0.000,B 0.000,C 90.000,E1 331.051} C_DIS
LIN {X 0.280,Y -503.352,Z 1332.638,A 0.000,B 0.000,C 90.000,E1 330.717} C_DIS
LIN {X 0.094,Y -502.121,Z 1332.637,A 0.000,B 0.000,C 90.000,E1 330.589} C_DIS
LIN {X -0.095,Y -500.315,Z 1332.636,A 0.000,B 0.000,C 90.000,E1 330.461} C_DIS
LIN {X 0.223,Y -474.384,Z 1332.626,A 0.000,B 0.000,C 90.000,E1 328.663} C_DIS
LIN {X 0.017,Y -451.219,Z 1332.616,A 0.000,B 0.000,C 90.000,E1 326.914} C_DIS
LIN {X -0.067,Y -430.040,Z 1332.606,A 0.000,B 0.000,C 90.000,E1 325.102} C_DIS
LIN {X 0.027,Y -409.358,Z 1332.595,A 0.000,B 0.000,C 90.000,E1 323.084} C_DIS
LIN {X -0.017,Y -390.658,Z 1332.584,A 0.000,B 0.000,C 90.000,E1 321.045} C_DIS
LIN {X 0.157,Y -375.926,Z 1332.574,A 0.000,B 0.000,C 90.000,E1 319.218} C_DIS
LIN {X 0.121,Y -375.916,Z 1332.574,A 0.000,B 0.000,C 90.000,E1 319.218} C_DIS
LIN {X 0.174,Y -378.219,Z 1332.563,A 0.000,B 0.000,C 90.000,E1 317.310} C_DIS
LIN {X 0.166,Y -383.907,Z 1332.531,A 0.000,B 0.000,C 90.000,E1 311.515} C_DIS
LIN {X -0.040,Y -384.874,Z 1332.527,A 0.000,B 0.000,C 90.000,E1 310.825} C_DIS
LIN {X -0.118,Y -390.577,Z 1332.495,A 0.000,B 0.000,C 90.000,E1 305.105} C_DIS
LIN {X -0.051,Y -391.070,Z 1332.493,A 0.000,B 0.000,C 90.000,E1 304.739} C_DIS
LIN {X -0.206,Y -391.414,Z 1332.491,A 0.000,B 0.000,C 90.000,E1 304.405} C_DIS
LIN {X 0.086,Y -396.794,Z 1332.459,A 0.000,B 0.000,C 90.000,E1 298.693} C_DIS
LIN {X -0.044,Y -397.110,Z 1332.458,A 0.000,B 0.000,C 90.000,E1 298.359} C_DIS
LIN {X 0.112,Y -401.577,Z 1332.426,A 0.000,B 0.000,C 90.000,E1 292.717} C_DIS
LIN {X 0.002,Y -404.637,Z 1332.395,A 0.000,B 0.000,C 90.000,E1 287.149} C_DIS
LIN {X -0.015,Y -404.754,Z 1332.393,A 0.000,B 0.000,C 90.000,E1 286.804} C_DIS
LIN {X -0.017,Y -406.086,Z 1332.364,A 0.000,B 0.000,C 90.000,E1 281.591} C_DIS
LIN {X -0.008,Y -406.104,Z 1332.363,A 0.000,B 0.000,C 90.000,E1 281.243} C_DIS
LIN {X 0.027,Y -405.674,Z 1332.334,A 0.000,B 0.000,C 90.000,E1 276.030} C_DIS
LIN {X 0.036,Y -405.300,Z 1332.330,A 0.000,B 0.000,C 90.000,E1 275.334} C_DIS
LIN {X 0.106,Y -403.511,Z 1332.305,A 0.000,B 0.000,C 90.000,E1 270.802} C_DIS
LIN {X 0.074,Y -403.302,Z 1332.303,A 0.000,B 0.000,C 90.000,E1 270.458} C_DIS
LIN {X -0.141,Y -398.954,Z 1332.272,A 0.000,B 0.000,C 90.000,E1 264.894} C_DIS
LIN {X 0.053,Y -393.127,Z 1332.242,A 0.000,B 0.000,C 90.000,E1 259.577} C_DIS
LIN {X 0.085,Y -392.859,Z 1332.240,A 0.000,B 0.000,C 90.000,E1 259.218} C_DIS
LIN {X 0.199,Y -386.018,Z 1332.213,A 0.000,B 0.000,C 90.000,E1 254.212} C_DIS
LIN {X 0.138,Y -385.291,Z 1332.208,A 0.000,B 0.000,C 90.000,E1 253.504} C_DIS
LIN {X 0.159,Y -384.812,Z 1332.207,A 0.000,B 0.000,C 90.000,E1 253.142} C_DIS
LIN {X -0.106,Y -378.004,Z 1332.182,A 0.000,B 0.000,C 90.000,E1 248.847} C_DIS
LIN {X 0.118,Y -376.260,Z 1332.174,A 0.000,B 0.000,C 90.000,E1 247.358} C_DIS
LIN {X -0.126,Y -374.991,Z 1332.170,A 0.000,B 0.000,C 90.000,E1 246.666} C_DIS
LIN {X -0.047,Y -368.452,Z 1332.148,A 0.000,B 0.000,C 90.000,E1 242.615} C_DIS
LIN {X 0.078,Y -366.094,Z 1332.138,A 0.000,B 0.000,C 90.000,E1 240.745} C_DIS
LIN {X 0.164,Y -359.232,Z 1332.115,A 0.000,B 0.000,C 90.000,E1 236.628} C_DIS
LIN {X 0.181,Y -355.888,Z 1332.100,A 0.000,B 0.000,C 90.000,E1 233.989} C_DIS
LIN {X -0.016,Y -348.827,Z 1332.075,A 0.000,B 0.000,C 90.000,E1 229.461} C_DIS
LIN {X 0.060,Y -346.211,Z 1332.062,A 0.000,B 0.000,C 90.000,E1 227.148} C_DIS
LIN {X -0.053,Y -345.726,Z 1332.060,A 0.000,B 0.000,C 90.000,E1 226.782} C_DIS
LIN {X 0.166,Y -344.127,Z 1332.054,A 0.000,B 0.000,C 90.000,E1 225.729} C_DIS
LIN {X 0.147,Y -344.135,Z 1332.054,A 0.000,B 0.000,C 90.000,E1 225.729} C_DIS
LIN {X -0.081,Y -359.772,Z 1332.041,A 0.000,B 0.000,C 90.000,E1 223.338} C_DIS
LIN {X 0.179,Y -376.032,Z 1332.028,A 0.000,B 0.000,C 90.000,E1 221.067} C_DIS
LIN {X 0.101,Y -393.188,Z 1332.017,A 0.000,B 0.000,C 90.000,E1 218.991} C_DIS
LIN {X -0.088,Y -412.316,Z 1332.005,A 0.000,B 0.000,C 90.000,E1 216.950} C_DIS
LIN {X 0.112,Y -433.472,Z 1331.994,A 0.000,B 0.000,C 90.000,E1 214.898} C_DIS
LIN {X -0.159,Y -444.139,Z 1331.989,A 0.000,B 0.000,C 90.000,E1 213.992} C_DIS
LIN {X -0.078,Y -445.857,Z 1331.987,A 0.000,B 0.000,C 90.000,E1 213.706} C_DIS
LIN {X -0.022,Y -447.212,Z 1331.985,A 0.000,B 0.000,C 90.000,E1 213.372} C_DIS
LIN {X 0.046,Y -448.263,Z 1331.984,A 0.000,B 0.000,C 90.000,E1 213.038} C_DIS
LIN {X -0.187,Y -449.836,Z 1331.980,A 0.000,B 0.000,C 90.000,E1 212.418} C_DIS
LIN {X -0.026,Y -451.030,Z 1331.976,A 0.000,B 0.000,C 90.000,E1 211.750} C_DIS
LIN {X -0.151,Y -452.321,Z 1331.971,A 0.000,B 0.000,C 90.000,E1 210.797} C_DIS
LIN {X 0.090,Y -454.038,Z 1331.962,A 0.000,B 0.000,C 90.000,E1 209.155} C_DIS
LIN {X -0.051,Y -457.722,Z 1331.946,A 0.000,B 0.000,C 90.000,E1 206.283} C_DIS
LIN {X 0.202,Y -460.516,Z 1331.935,A 0.000,B 0.000,C 90.000,E1 204.335} C_DIS
LIN {X -0.082,Y -463.072,Z 1331.925,A 0.000,B 0.000,C 90.000,E1 202.461} C_DIS
LIN {X 0.009,Y -465.179,Z 1331.916,A 0.000,B 0.000,C 90.000,E1 200.865} C_DIS
LIN {X 0.078,Y -467.560,Z 1331.905,A 0.000,B 0.000,C 90.000,E1 198.960} C_DIS
LIN {X -0.055,Y -469.480,Z 1331.897,A 0.000,B 0.000,C 90.000,E1 197.402} C_DIS
LIN {X 0.091,Y -470.675,Z 1331.891,A 0.000,B 0.000,C 90.000,E1 196.441} C_DIS
LIN {X -0.110,Y -472.453,Z 1331.883,A 0.000,B 0.000,C 90.000,E1 194.898} C_DIS
LIN {X 0.180,Y -474.219,Z 1331.874,A 0.000,B 0.000,C 90.000,E1 193.300} C_DIS
LIN {X -0.232,Y -476.332,Z 1331.864,A 0.000,B 0.000,C 90.000,E1 191.478} C_DIS
LIN {X -0.073,Y -478.154,Z 1331.855,A 0.000,B 0.000,C 90.000,E1 189.905} C_DIS
LIN {X 0.043,Y -479.877,Z 1331.846,A 0.000,B 0.000,C 90.000,E1 188.341} C_DIS
LIN {X 0.070,Y -480.845,Z 1331.841,A 0.000,B 0.000,C 90.000,E1 187.409} C_DIS
LIN {X -0.160,Y -481.977,Z 1331.834,A 0.000,B 0.000,C 90.000,E1 186.201} C_DIS
LIN {X 0.112,Y -483.007,Z 1331.828,A 0.000,B 0.000,C 90.000,E1 184.935} C_DIS
LIN {X 0.101,Y -483.729,Z 1331.822,A 0.000,B 0.000,C 90.000,E1 184.012} C_DIS
LIN {X 0.058,Y -484.186,Z 1331.817,A 0.000,B 0.000,C 90.000,E1 183.094} C_DIS
LIN {X -0.177,Y -484.625,Z 1331.810,A 0.000,B 0.000,C 90.000,E1 181.892} C_DIS
LIN {X -0.210,Y -484.846,Z 1331.805,A 0.000,B 0.000,C 90.000,E1 180.974} C_DIS
LIN {X 0.233,Y -484.894,Z 1331.800,A 0.000,B 0.000,C 90.000,E1 180.000} C_DIS
LIN {X 0.015,Y -484.757,Z 1331.793,A 0.000,B 0.000,C 90.000,E1 178.797} C_DIS
LIN {X -0.016,Y -484.447,Z 1331.788,A 0.000,B 0.000,C 90.000,E1 177.879} C_DIS
LIN {X -0.070,Y -484.013,Z 1331.783,A 0.000,B 0.000,C 90.000,E1 176.963} C_DIS
LIN {X -0.109,Y -483.306,Z 1331.778,A 0.000,B 0.000,C 90.000,E1 176.045} C_DIS
LIN {X -0.116,Y -482.347,Z 1331.773,A 0.000,B 0.000,C 90.000,E1 175.122} C_DIS
LIN {X 0.157,Y -480.710,Z 1331.766,A 0.000,B 0.000,C 90.000,E1 173.856} C_DIS
LIN {X -0.081,Y -478.558,Z 1331.759,A 0.000,B 0.000,C 90.000,E1 172.648} C_DIS
LIN {X -0.234,Y -477.934,Z 1331.757,A 0.000,B 0.000,C 90.000,E1 172.356} C_DIS
LIN {X 0.176,Y -475.490,Z 1331.752,A 0.000,B 0.000,C 90.000,E1 171.376} C_DIS
LIN {X -0.144,Y -473.679,Z 1331.749,A 0.000,B 0.000,C 90.000,E1 170.792} C_DIS
LIN {X -0.197,Y -471.948,Z 1331.746,A 0.000,B 0.000,C 90.000,E1 170.330} C_DIS
LIN {X -0.077,Y -469.408,Z 1331.743,A 0.000,B 0.000,C 90.000,E1 169.690} C_DIS
LIN {X 0.206,Y -468.021,Z 1331.741,A 0.000,B 0.000,C 90.000,E1 169.342} C_DIS
LIN {X 0.011,Y -463.651,Z 1331.737,A 0.000,B 0.000,C 90.000,E1 168.578} C_DIS
LIN {X 0.063,Y -459.779,Z 1331.733,A 0.000,B 0.000,C 90.000,E1 167.937} C_DIS
LIN {X -0.118,Y -450.620,Z 1331.725,A 0.000,B 0.000,C 90.000,E1 166.520} C_DIS
LIN {X 0.140,Y -443.305,Z 1331.719,A 0.000,B 0.000,C 90.000,E1 165.353} C_DIS
LIN {X 0.252,Y -430.133,Z 1331.707,A 0.000,B 0.000,C 90.000,E1 163.196} C_DIS
LIN {X -0.173,Y -429.168,Z 1331.706,A 0.000,B 0.000,C 90.000,E1 163.087} C_DIS
LIN {X -0.060,Y -425.825,Z 1331.701,A 0.000,B 0.000,C 90.000,E1 162.236} C_DIS
LIN {X 0.069,Y -425.377,Z 1331.698,A 0.000,B 0.000,C 90.000,E1 161.529} C_DIS
LIN {X 0.176,Y -426.034,Z 1331.696,A 0.000,B 0.000,C 90.000,E1 161.275} C_DIS
LIN {X 0.133,Y -426.083,Z 1331.696,A 0.000,B 0.000,C 90.000,E1 161.275} C_DIS
LIN {X 0.088,Y -427.735,Z 1331.695,A 0.000,B 0.000,C 90.000,E1 161.094} C_DIS
LIN {X 0.038,Y -429.503,Z 1331.694,A 0.000,B 0.000,C 90.000,E1 160.859} C_DIS
LIN {X -0.017,Y -433.678,Z 1331.692,A 0.000,B 0.000,C 90.000,E1 160.477} C_DIS
LIN {X -0.157,Y -445.797,Z 1331.686,A 0.000,B 0.000,C 90.000,E1 159.518} C_DIS
LIN {X 0.010,Y -459.748,Z 1331.680,A 0.000,B 0.000,C 90.000,E1 158.411} C_DIS
LIN {X 0.218,Y -469.052,Z 1331.676,A 0.000,B 0.000,C 90.000,E1 157.667} C_DIS
LIN {X -0.156,Y -476.699,Z 1331.673,A 0.000,B 0.000,C 90.000,E1 157.102} C_DIS
LIN {X -0.258,Y -481.159,Z 1331.671,A 0.000,B 0.000,C 90.000,E1 156.741} C_DIS
LIN {X 0.132,Y -487.068,Z 1331.668,A 0.000,B 0.000,C 90.000,E1 156.177} C_DIS
LIN {X -0.144,Y -494.245,Z 1331.664,A 0.000,B 0.000,C 90.000,E1 155.537} C_DIS
LIN {X 0.128,Y -498.415,Z 1331.662,A 0.000,B 0.000,C 90.000,E1 155.101} C_DIS
LIN {X -0.050,Y -506.562,Z 1331.657,A 0.000,B 0.000,C 90.000,E1 154.280} C_DIS
LIN {X -0.057,Y -512.788,Z 1331.653,A 0.000,B 0.000,C 90.000,E1 153.589} C_DIS
LIN {X 0.148,Y -516.548,Z 1331.651,A 0.000,B 0.000,C 90.000,E1 153.127} C_DIS
LIN {X 0.170,Y -521.239,Z 1331.648,A 0.000,B 0.000,C 90.000,E1 152.538} C_DIS
LIN {X -0.017,Y -525.381,Z 1331.644,A 0.000,B 0.000,C 90.000,E1 151.975} C_DIS
LIN {X 0.071,Y -529.001,Z 1331.641,A 0.000,B 0.000,C 90.000,E1 151.385} C_DIS
LIN {X 0.038,Y -532.719,Z 1331.637,A 0.000,B 0.000,C 90.000,E1 150.667} C_DIS
LIN {X 0.033,Y -535.612,Z 1331.633,A 0.000,B 0.000,C 90.000,E1 149.950} C_DIS
LIN {X -0.272,Y -537.573,Z 1331.630,A 0.000,B 0.000,C 90.000,E1 149.410} C_DIS
LIN {X -0.101,Y -540.033,Z 1331.625,A 0.000,B 0.000,C 90.000,E1 148.535} C_DIS
LIN {X 0.100,Y -542.166,Z 1331.620,A 0.000,B 0.000,C 90.000,E1 147.661} C_DIS
LIN {X -0.155,Y -543.403,Z 1331.617,A 0.000,B 0.000,C 90.000,E1 147.120} C_DIS
LIN {X 0.108,Y -545.447,Z 1331.611,A 0.000,B 0.000,C 90.000,E1 145.960} C_DIS
LIN {X 0.218,Y -546.656,Z 1331.606,A 0.000,B 0.000,C 90.000,E1 145.102} C_DIS
LIN {X 0.076,Y -547.862,Z 1331.600,A 0.000,B 0.000,C 90.000,E1 143.989} C_DIS
LIN {X 0.271,Y -548.755,Z 1331.594,A 0.000,B 0.000,C 90.000,E1 142.844} C_DIS
LIN {X 0.203,Y -550.000,Z 1331.583,A 0.000,B 0.000,C 90.000,E1 140.884} C_DIS
LIN {X 0.086,Y -551.558,Z 1331.572,A 0.000,B 0.000,C 90.000,E1 138.933} C_DIS
LIN {X -0.066,Y -552.161,Z 1331.570,A 0.000,B 0.000,C 90.000,E1 138.528} C_DIS
LIN {X -0.223,Y -552.775,Z 1331.569,A 0.000,B 0.000,C 90.000,E1 138.405} C_DIS
LIN {X -0.065,Y -553.882,Z 1331.567,A 0.000,B 0.000,C 90.000,E1 138.038} C_DIS
LIN {X 0.138,Y -553.915,Z 1331.567,A 0.000,B 0.000,C 90.000,E1 138.000} C_DIS
LIN {X 0.095,Y -553.924,Z 1331.567,A 0.000,B 0.000,C 90.000,E1 138.000} C_DIS
LIN {X 0.149,Y -555.841,Z 1331.566,A 0.000,B 0.000,C 90.000,E1 137.877} C_DIS
LIN {X 0.001,Y -567.614,Z 1331.564,A 0.000,B 0.000,C 90.000,E1 137.553} C_DIS
LIN {X 0.332,Y -574.006,Z 1331.563,A 0.000,B 0.000,C 90.000,E1 137.310} C_DIS
